      OPN   #DB_VI;  // Abro el DB a resetear
      LAR1  P##PunteroDBVI;  // Preparar el Puntero Any
      L     B#16#10;  // ID de Sintasis
      T     LB [AR1, P#0.0];
      L     B#16#2;  // Tipo de Datos
      T     LB [AR1, P#1.0];
      L     DBLG;  // Longitud del DB
      T     LW [AR1, P#2.0];
      L     DBNO;  // Numero de DB
      T     LW [AR1, P#4.0];
      L     0;
      SLW   3;
      T     LD [AR1, P#6.0];
      L     B#16#84;  // Indico el tipo DB
      T     LB [AR1, P#6.0];

      L     0;  // Que rellenar en el DB
      T     #ByteTMP;
      CALL  FILL
      ( BVAL    := #ByteTMP,
        RET_VAL := #ReturnValor,
        BLK     := #PunteroDBVI
      );  // Reseteo el DB


/////////////////////////////////////////////////////////////////////////////
// --- Reseteo - Estado del Vehiculo Inteligente

      L     0;  // Reseteo del Estado del VI
      T     #ByteTMP;
      CALL  FILL
      ( BVAL    := #ByteTMP,
        RET_VAL := #ReturnValor,
        BLK     := "DB900_Estado_Mesas".EstadoVI[#Mesa]
      );

/////////////////////////////////////////////////////////////////////////////
// --- No hay más que resetar
      JU    SistemaReset_Gestion;


/////////////////////////////////////////////////////////////////////////////
/////////////////////////////////////////////////////////////////////////////
/////////////////////////////////////////////////////////////////////////////
/////////////////////////////////////////////////////////////////////////////
// --- Reset Imposible

ResetImposible:NOP   0;
      SET;
      S     "DB840_Emision".DispoMesa[#Mesa].Protocolo.ResetNOK;  // Activacion de Reset Imposible
      R     "DB840_Emision".DispoMesa[#Mesa].Protocolo.ResetOK;  // DesActivacion de Reset OK
      R     "DB840_Emision".DispoMesa[#Mesa].Protocolo.Reset_Realizandose;  // Desactivar el Reset
      R     "DB831_Mesas".Mesas[#Mesa].Memorias.M_ResetParcial;  // Memo Reset Parcial
      R     "DB831_Mesas".Mesas[#Mesa].Memorias.M_ResetTotal;  // Memo Reset Total

      JU    SistemaReset_Gestion;


/////////////////////////////////////////////////////////////////////////////
/////////////////////////////////////////////////////////////////////////////
/////////////////////////////////////////////////////////////////////////////
/////////////////////////////////////////////////////////////////////////////
// --- Gestion de Reset
SistemaReset_Gestion:NOP   0;
      SET;
      AN    "DB840_Emision".DispoMesa[#Mesa].Protocolo.Reset_Realizandose;
      JC    SistemaReset_Fin;  // Hay Reset en el Sistema ?

      SET;
      AN    #EstadoZona.Resetear_CBx;  // Por la Zona
      AN    #EstadoZona.PerReset_CBx;
      AN    "DB841_Recepcion".DispoMesa[#Mesa].Protocolo.Reset;  // Por la Orden de la Mesa
      AN    "DB843_RecepcionPantalla".Mesa[#Mesa].Reset;  // Por la Orden de la Pantalla
      A     "DB841_Recepcion".DispoMesa[#Mesa].Protocolo.EmiOK;  // Avisado el JdT ?
      JCN   SistemaReset_Continuar;


/////////////////////////////////////////////////////////////////////////////
// --- Reset Finalizazado
      SET;
      R     "DB840_Emision".DispoMesa[#Mesa].Protocolo.Reset_Realizandose;
      R     "DB831_Mesas".Mesas[#Mesa].Memorias.M_ResetParcial;  // Memo Reset Parcial
      R     "DB831_Mesas".Mesas[#Mesa].Memorias.M_ResetTotal;  // Memo Reset Total -


/////////////////////////////////////////////////////////////////////////////
/////////////////////////////////////////////////////////////////////////////
/////////////////////////////////////////////////////////////////////////////
// --- Continuar con el Reset

SistemaReset_Continuar:NOP   0;
      SET;
      A     #FinResetTMP;  // Fin de Reset del VI ?
      S     "DB840_Emision".DispoMesa[#Mesa].Protocolo.ResetOK;  // Aviso de Fin de Reset


// --- Si no llega el Fin de Reset en un tiempo determinado
      SET;
      AN    #FinResetTMP;  // No, Fin de Reset del VI ?
      AN    "DB840_Emision".DispoMesa[#Mesa].Protocolo.ResetOK;  // No, Aviso de Fin de Reset
      AN    "DB840_Emision".DispoMesa[#Mesa].Protocolo.ResetNOK;  // No, Aviso de Fin de Reset
      A     #TIM_FinReset_OK;  // Se cumplido el tiempo de Espera
      A     "DB840_Emision".DispoMesa[#Mesa].Protocolo.Reset_Realizandose;  // Reset Realizandose
      JC    ResetImposible;  // Activar reset imposible


// --- Finalizado
      JU    SistemaReset_Fin;  // Ir al Final de Reset


/////////////////////////////////////////////////////////////////////////////
/////////////////////////////////////////////////////////////////////////////
/////////////////////////////////////////////////////////////////////////////
/////////////////////////////////////////////////////////////////////////////
// --- Fin del sistema de Reset

SistemaReset_Fin:NOP   0;
      SET;
      AN    "DB840_Emision".DispoMesa[#Mesa].Protocolo.Reset_Realizandose;
      R     "DB840_Emision".DispoMesa[#Mesa].Protocolo.ResetOK;  // No Aviso de Fin de Reset

      SET;
      A     "DB840_Emision".DispoMesa[#Mesa].Protocolo.ResetNOK;
      A     "DB841_Recepcion".DispoMesa[#Mesa].Protocolo.EmiOK;
      R     "DB840_Emision".DispoMesa[#Mesa].Protocolo.ResetNOK;  // Desactivacion de Reset Imposible



NETWORK
TITLE = ---- Presencias de la Mesa en el Reset
/////////////////////////////////////////////////////////////////////////////
// --- Presencias de la Mesa en el Reset
      SET;
      A     "DB840_Emision".Mesa[#Mesa].Protocolo.PresNormal;
      A     "DB900_Estado_Mesas".EstadoVI[#Mesa].Etapas_Reset;
      =     "DB840_Emision".Mesa[#Mesa].Protocolo.PresReset;  // Presencia de Reset

/////////////////////////////////////////////////////////////////////////////
// --- Comprobar que se esta haciendo Reset
      SET;
      AN    "DB840_Emision".DispoMesa[#Mesa].Protocolo.Reset_Realizandose;
      JC    Final_PresenciaEnReset;

/////////////////////////////////////////////////////////////////////////////
// --- Flanco en el Reset
      SET;
      A     "DB840_Emision".Mesa[#Mesa].Protocolo.PresReset;  // Emision del VI
      FP    "DB831_Mesas".Mesas[#Mesa].Memorias.MFL_PresReset;
      =     #FlancoPresReset;

/////////////////////////////////////////////////////////////////////////////
// --- Creacion de UT en Reset Total
      SET;
      A     "DB831_Mesas".Mesas[#Mesa].Memorias.M_ResetTotal;  // Memo Reset Total
      A     #FlancoPresReset;
      JCN   Final_PresenciaEnReset;

// Creo una nueva UT
      CALL  "FC723_InsertarUT_EnMesa"
      ( MesaActual := #Mesa,
        NumeroUT   := #NumeroUT
      );

      JU    Final_PresenciaEnReset;

/////////////////////////////////////////////////////////////////////////////
Final_PresenciaEnReset:NOP   0;



NETWORK
TITLE = Gestion del Control de Paro Blando
/////////////////////////////////////////////////////////////////////////////
// --- Flanco de la Activacion de la Gestion del Paro Blando
      SET;
      A     "DB841_Recepcion".DispoMesa[#Mesa].Protocolo.ParoBlando;  // Por la Orden de Mesa
      O     "DB843_RecepcionPantalla".Mesa[#Mesa].ParoBlando;  // Por la Orden de la Pantalla
      FP    "DB831_Mesas".Mesas[#Mesa].Memorias.MFL_ParoBlando;  // Memo Paro Blando - Pos: 22.7
      =     #FlancoParoBlando;

      SET;
      A     #FinParoBlando;  // No hace caso si no hay Paro Blando
      A     "DB900_Estado_Mesas".EstadoVI[#Mesa].Paro_Blando;
      A     "DB840_Emision".DispoMesa[#Mesa].Protocolo.ParoBlando_Realizandose;
      =     #FinParoBlandoTMP;


/////////////////////////////////////////////////////////////////////////////
// --- Activacion de la Gestion del Paro Blando

      AN    #FlancoParoBlando;
      JC    SistemaParoBlando_Gestion;  // Hay que realizar el Paro Blando ?

      SET;
      S     "DB840_Emision".DispoMesa[#Mesa].Protocolo.ParoBlando_Realizandose;

      JU    SistemaParoBlando_Gestion;

/////////////////////////////////////////////////////////////////////////////
/////////////////////////////////////////////////////////////////////////////
/////////////////////////////////////////////////////////////////////////////
/////////////////////////////////////////////////////////////////////////////
// --- Paro Blando Imposible

ParoBlandoImposible:NOP   0;
      S     "DB840_Emision".DispoMesa[#Mesa].Protocolo.ParoBlandoNOK;  // Activacion de Paro Blando Imposible
      R     "DB840_Emision".DispoMesa[#Mesa].Protocolo.ParoBlandoOK;  // DesActivacion de Paro Blando OK

      R     "DB840_Emision".DispoMesa[#Mesa].Protocolo.ParoBlando_Realizandose;  // Acabado Paro Blando
      R     "DB840_Emision".DispoMesa[#Mesa].Protocolo.Marcha;  // Se pasa a Paro
      S     "DB840_Emision".DispoMesa[#Mesa].Protocolo.Paro;

      JU    SistemaParoBlando_Gestion;

/////////////////////////////////////////////////////////////////////////////
/////////////////////////////////////////////////////////////////////////////
/////////////////////////////////////////////////////////////////////////////
// --- Gestion del Paro Blando

SistemaParoBlando_Gestion:NOP   0;
      SET;
      AN    "DB840_Emision".DispoMesa[#Mesa].Protocolo.ParoBlando_Realizandose;
      JC    SistemaParoBlando_Fin;  // Hay Paro Blando en el Sistema ?

      SET;
      AN    "DB841_Recepcion".DispoMesa[#Mesa].Protocolo.ParoBlando;  // Por la Orden de la Mesa
      AN    "DB843_RecepcionPantalla".Mesa[#Mesa].ParoBlando;  // Por la Orden de la Pantalla
      A     "DB841_Recepcion".DispoMesa[#Mesa].Protocolo.EmiOK;  // Avisado el JdT ?
      JCN   SistemaParoBlando_Continuar;


/////////////////////////////////////////////////////////////////////////////
/////////////////////////////////////////////////////////////////////////////
/////////////////////////////////////////////////////////////////////////////
// --- Fin de Paro Blando Finalizado

      SET;
      R     "DB840_Emision".DispoMesa[#Mesa].Protocolo.ParoBlando_Realizandose;  // Acabado Paro Blando
      R     "DB840_Emision".DispoMesa[#Mesa].Protocolo.Marcha;  // Se pasa a Paro
      S     "DB840_Emision".DispoMesa[#Mesa].Protocolo.Paro;

/////////////////////////////////////////////////////////////////////////////
/////////////////////////////////////////////////////////////////////////////
/////////////////////////////////////////////////////////////////////////////
// --- Continuar con el Paro Blando
SistemaParoBlando_Continuar:NOP   0;

      SET;
      A     #FinParoBlandoTMP;  // Fin de ParoBlando del VI ?
      S     "DB840_Emision".DispoMesa[#Mesa].Protocolo.ParoBlandoOK;  // Aviso de Fin de Paro Blando

// --- Si no llega el Fin de Paro Blando en un tiempo determinado
      SET;
      AN    #FinParoBlandoTMP;  // No, Fin de Paro Blando del VI ?
      AN    "DB840_Emision".DispoMesa[#Mesa].Protocolo.ParoBlandoOK;  // No, Aviso de Fin de Paro Blando
      AN    "DB840_Emision".DispoMesa[#Mesa].Protocolo.ParoBlandoNOK;  // No, Aviso de Fin de Paro Blando
      A     #TIM_FinParoBlando_OK;  // Se cumplido el tiempo de Espera
      A     "DB840_Emision".DispoMesa[#Mesa].Protocolo.ParoBlando_Realizandose;  // Paro Blando Realizandose
      JC    ParoBlandoImposible;  // Activar Paro Blando imposible


/////////////////////////////////////////////////////////////////////////////
// --- Fin del sistema de Paro Blando

SistemaParoBlando_Fin:NOP   0;
      SET;
      AN    "DB840_Emision".DispoMesa[#Mesa].Protocolo.ParoBlando_Realizandose;
      R     "DB840_Emision".DispoMesa[#Mesa].Protocolo.ParoBlandoOK;  // No Aviso de Fin de Paro Blando

      SET;
      A     "DB840_Emision".DispoMesa[#Mesa].Protocolo.ParoBlandoNOK;
      A     "DB841_Recepcion".DispoMesa[#Mesa].Protocolo.EmiOK;
      R     "DB840_Emision".DispoMesa[#Mesa].Protocolo.ParoBlandoNOK;  // Desactivacion de Paro Blando Imposible



NETWORK
TITLE = Gestion del Control de Error de la Mesa
/////////////////////////////////////////////////////////////////////////////
// --- Calculo del Error de la Mesa

      AN    "DB900_Estado_Mesas".EstadoVI[#Mesa].Error_Mx;
      JC    NoErrorEnMesa;


/////////////////////////////////////////////////////////////////////////////
      L     #Mesa;  // Puntero al DB de Estado VI
      L     "CTE_Long_VIMesa";  // Longitud de la UDT 20
      *D;
      SLD   3;
      T     #P_EstadoVI;

      L     "CTE_NDB_EstadoVIMesa";  // DB de Estado VI
      T     #DBEstadoVI;

      L     #P_EstadoVI;  // Punteros
      L     P#2.0;
      +D;
      LAR2;
      T     #PunteroDBTMP;  // Offset dentro del DB

      OPN   DB [#DBEstadoVI];
Bucle_ErrorVI:NOP   0;
      A     DBX [AR2, P#0.0];
      JC    EncontradoErrorEnMesa;

      +AR2  P#0.1;
      JU    Bucle_ErrorVI;


/////////////////////////////////////////////////////////////////////////////
// --- Con Error
EncontradoErrorEnMesa:NOP   0;
      TAR2;
      L     #PunteroDBTMP;
      -D;
      L     1;
      +D;
      T     #NumeroErrorVI;
      T     "DB840_Emision".DispoMesa[#Mesa].Error;

      L     #NumeroErrorVI;
      T     #CodigoErrorMesa;
      T     "DB861_FIFO_Errores".Mesas[#Mesa];

      JU    FinGestion_Error;


/////////////////////////////////////////////////////////////////////////////
// --- Sin Error
NoErrorEnMesa:NOP   0;
      L     0;
      T     #CodigoErrorMesa;
      T     "DB840_Emision".DispoMesa[#Mesa].Error;
      T     "DB861_FIFO_Errores".Mesas[#Mesa];

      JU    FinGestion_Error;


/////////////////////////////////////////////////////////////////////////////
// --- Rearme y Activacion del Error
FinGestion_Error:NOP   0;
      SET;
      A     #EstadoZona.Rearme_CBx;  // Por la Zona
      O     #RearmeError;  // Manualmente (Exterior)
      O     "DB841_Recepcion".DispoMesa[#Mesa].Protocolo.Rearme;  // Por la Orden
      O     "DB843_RecepcionPantalla".Mesa[#Mesa].Rearme;  // Por la Orden de Pantalla
      =     "DB902_Estado_ZonaMesa".EstadoMesas[#Mesa].Rearme_CBx;

      SET;
      A     "DB900_Estado_Mesas".EstadoVI[#Mesa].Error_Mx;
      =     "DB840_Emision".DispoMesa[#Mesa].Protocolo.Error;  // Esta en Error el VI



REGION Network 10: Cierre del Protocolo de la Mesa
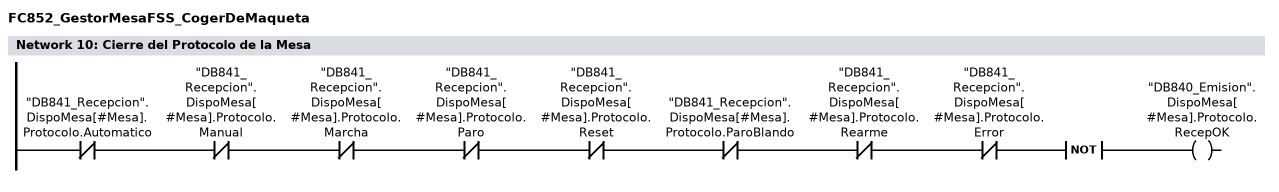
   RUNG wire#powerrail
      I_Contact( "DB841_Recepcion".DispoMesa[#Mesa].Protocolo.Automatico )
      I_Contact( "DB841_Recepcion".DispoMesa[#Mesa].Protocolo.Manual )
      I_Contact( "DB841_Recepcion".DispoMesa[#Mesa].Protocolo.Marcha )
      I_Contact( "DB841_Recepcion".DispoMesa[#Mesa].Protocolo.Paro )
      I_Contact( "DB841_Recepcion".DispoMesa[#Mesa].Protocolo.Reset )
      I_Contact( "DB841_Recepcion".DispoMesa[#Mesa].Protocolo.ParoBlando )
      I_Contact( "DB841_Recepcion".DispoMesa[#Mesa].Protocolo.Rearme )
      I_Contact( "DB841_Recepcion".DispoMesa[#Mesa].Protocolo.Error )
      Not()
      Coil( "DB840_Emision".DispoMesa[#Mesa].Protocolo.RecepOK )
   END_RUNG
   // the same network as SCL:
   "DB840_Emision".DispoMesa[#Mesa].Protocolo.RecepOK := NOT (NOT "DB841_Recepcion".DispoMesa[#Mesa].Protocolo.Automatico AND NOT "DB841_Recepcion".DispoMesa[#Mesa].Protocolo.Manual AND NOT "DB841_Recepcion".DispoMesa[#Mesa].Protocolo.Marcha AND NOT "DB841_Recepcion".DispoMesa[#Mesa].Protocolo.Paro AND NOT "DB841_Recepcion".DispoMesa[#Mesa].Protocolo.Reset AND NOT "DB841_Recepcion".DispoMesa[#Mesa].Protocolo.ParoBlando AND NOT "DB841_Recepcion".DispoMesa[#Mesa].Protocolo.Rearme AND NOT "DB841_Recepcion".DispoMesa[#Mesa].Protocolo.Error);
END_REGION

NETWORK
TITLE = Cierre del Protocolo de la Pantalla
/////////////////////////////////////////////////////////////////////////////
// --- Cierre del protocolo de las ordenes de la Pantalla
// --- Doy por tratada la Orden

      L     0;  // Que rellenar en el DB
      T     #ByteTMP;

      CALL  FILL
      ( BVAL    := #ByteTMP,
        RET_VAL := #ReturnValor,
        BLK     := "DB843_RecepcionPantalla".Mesa[#Mesa]
      );  // Reseteo el la zona temp



NETWORK
TITLE = Actualizacion del Estado para el Vehiculo Inteligente
/////////////////////////////////////////////////////////////////////////////
// --- Trasvase - Estado de la Mesa para VI

      A     "DB840_Emision".DispoMesa[#Mesa].Protocolo.Error;
      =     "DB902_Estado_ZonaMesa".EstadoMesas[#Mesa].Error_CBx;
      A     "DB840_Emision".DispoMesa[#Mesa].Protocolo.Marcha;
      =     "DB902_Estado_ZonaMesa".EstadoMesas[#Mesa].Marcha_CBx;
      A     "DB840_Emision".DispoMesa[#Mesa].Protocolo.Paro;
      =     "DB902_Estado_ZonaMesa".EstadoMesas[#Mesa].Paro_CBx;

      A     "DB840_Emision".DispoMesa[#Mesa].Protocolo.Automatico;
      =     "DB902_Estado_ZonaMesa".EstadoMesas[#Mesa].Automatico_CBx;
      A     "DB840_Emision".DispoMesa[#Mesa].Protocolo.Manual;
      =     "DB902_Estado_ZonaMesa".EstadoMesas[#Mesa].Manual_CBx;

      A     #FlancoReset;
      =     "DB902_Estado_ZonaMesa".EstadoMesas[#Mesa].Resetear_CBx;
      A     "DB840_Emision".DispoMesa[#Mesa].Protocolo.Reset_Realizandose;
      =     "DB902_Estado_ZonaMesa".EstadoMesas[#Mesa].PerReset_CBx;

      A     "DB840_Emision".DispoMesa[#Mesa].Protocolo.ParoBlando_Realizandose;
      =     "DB902_Estado_ZonaMesa".EstadoMesas[#Mesa].ParoBlando_CBx;



NETWORK
TITLE = Control de Error de Mesa por Orden del JdT
/////////////////////////////////////////////////////////////////////////////
/////////////////////////////////////////////////////////////////////////////
// --- Rearme de Errores Generados
// --- Borrado errores Mesa --> JdT

      SET;
      A     #EstadoZona.Rearme_CBx;  // Por la Zona
      O     #RearmeError;  // Manualmente (Exterior)
      O     "DB841_Recepcion".DispoMesa[#Mesa].Protocolo.Rearme;  // Por la Orden
      O     "DB843_RecepcionPantalla".Mesa[#Mesa].Rearme;  // Por la Orden de Pantalla
      JCN   NoRearme_ErrorJdT;

      SET;
      R     "DB900_Estado_Mesas".EstadoVI[#Mesa].Err_EnviadoPorJDT;  // Error Enviado por JDT
      R     "DB900_Estado_Mesas".EstadoVI[#Mesa].Error_Mx;  // Error de Mesa


NoRearme_ErrorJdT:NOP   0;


/////////////////////////////////////////////////////////////////////////////
/////////////////////////////////////////////////////////////////////////////
// --- Mirar errores Mesa --> JdT

      SET;
      AN    "DB841_Recepcion".DispoMesa[#Mesa].Protocolo.Error;
      JC    NoRecibido_ErrorJdT;

      SET;
      S     "DB900_Estado_Mesas".EstadoVI[#Mesa].Err_EnviadoPorJDT;  // Error Enviado por JDT
      S     "DB900_Estado_Mesas".EstadoVI[#Mesa].Error_Mx;  // Error de Mesa

NoRecibido_ErrorJdT:NOP   0;



NETWORK
TITLE = Control de Errores entre la Mesa y el Tracking
/////////////////////////////////////////////////////////////////////////////
/////////////////////////////////////////////////////////////////////////////
/////////////////////////////////////////////////////////////////////////////
// --- Rearme de Errores Generados
// --- Borrado errores Mesa --> Tracking

      SET;
      A     #EstadoZona.Rearme_CBx;  // Por la Zona
      O     #RearmeError;  // Manualmente (Exterior)
      O     "DB841_Recepcion".DispoMesa[#Mesa].Protocolo.Rearme;  // Por la Orden
      O     "DB843_RecepcionPantalla".Mesa[#Mesa].Rearme;  // Por la Orden de Pantalla
      JCN   NoRearme_ErrorTracking;

      SET;
      R     "DB900_Estado_Mesas".EstadoVI[#Mesa].Err_DatosPLC;  // Error Datos del PLC
      R     "DB900_Estado_Mesas".EstadoVI[#Mesa].Error_Mx;  // Error de Mesa


NoRearme_ErrorTracking:NOP   0;


/////////////////////////////////////////////////////////////////////////////
/////////////////////////////////////////////////////////////////////////////
/////////////////////////////////////////////////////////////////////////////
// --- Listado de Errores implementados:
// ---     * Mesa Vacia con existencia de una UT
// ---     * Mesa Ocupada sin existencia de una UT

      CALL  "FC870_MesaSinUT"
      ( Mesa  := #Mesa,
        SinUT := #SinUT_EnMesa
      );

      SET;
      AN    "DB850_DefinicionMesas".Mesa[#Mesa].ConfigMesa.SinErrorDeDatosVacia;
      A     "DB840_Emision".DispoMesa[#Mesa].Protocolo.Marcha;
      AN    "DB840_Emision".DispoMesa[#Mesa].Protocolo.Error;
      A     "DB900_Estado_Mesas".EstadoVI[#Mesa].Etapa_Vacia;
      AN    #SinUT_EnMesa;
      =     #ErrorMesaVacia;

      SET;
      AN    "DB850_DefinicionMesas".Mesa[#Mesa].ConfigMesa.SinErrorDeDatosCargada;
      A     "DB840_Emision".DispoMesa[#Mesa].Protocolo.Marcha;
      AN    "DB840_Emision".DispoMesa[#Mesa].Protocolo.Error;
      A     "DB900_Estado_Mesas".EstadoVI[#Mesa].Etapa_Cargada;
      A     #SinUT_EnMesa;
      =     #ErrorMesaOcupada;

      SET;
      A     #ErrorMesaVacia;
      O     #ErrorMesaOcupada;
      =     #ActivarTMPErrorMesa;


/////////////////////////////////////////////////////////////////////////////
// ---     * Esperar tiempo antes de activar el Error

      CALL  "FC899_TMP"
      ( Temporizar     := #ActivarTMPErrorMesa,
        Valor_Tiempo   := 20,
        Base_tiempo_ms := 1000,
        Tiempo_OK      := #TIM_ErrorMesa_OK,
        Valor_Actual   := "DB831_Mesas".Mesas[#Mesa].TMP_ErrorDatos
      );


/////////////////////////////////////////////////////////////////////////////
// --- Mirar errores Mesa --> Tracking
      SET;
      AN    #TIM_ErrorMesa_OK;
      JC    NoExiste_ErrorTracking;

      SET;
      S     "DB900_Estado_Mesas".EstadoVI[#Mesa].Err_DatosPLC;  // Error Datos del PLC
      S     "DB900_Estado_Mesas".EstadoVI[#Mesa].Error_Mx;  // Error de Mesa

NoExiste_ErrorTracking:NOP   0;



NETWORK
TITLE = Cambio de Mesa o creación de la UT -- DIstribucion
// Realiza:
//  - Gestion de la realización del cambio de Mesa de la UT
//  - Creación de la UT nueva
/////////////////////////////////////////////////////////////////////////////
// --- Distribución de lo que se HARA ? y CUANDO ?
/////////////////////////////////////////////////////////////////////////////
// --- Entrada de la UT por E0
// --- Entrada de la UT por E1
// --- Entrada de la UT por E2
// --- Entrada de la UT por E3
// --- Entrada de la UT por E4
// ---
// --- Nota: Hay que identificar en cada entrada dos casos:
// ---       Cuando cambia de Mesa - Codigo 11
// ---       Cuando se crea la UT  - Codigo 12
/////////////////////////////////////////////////////////////////////////////

      SET;
      A     #TransferirUT;  // Orden de Transferir la UT
      FP    "DB831_Mesas".Mesas[#Mesa].Memorias.MFL_TransferirUT;
      =     #FlancoTransferirUT;

      SET;
      AN    #FlancoTransferirUT;
      JC    FinalControlUTs_EnMesa;


/////////////////////////////////////////////////////////////////////////////
/////////////////////////////////////////////////////////////////////////////
// ---                     DISTRIBUCION
/////////////////////////////////////////////////////////////////////////////
/////////////////////////////////////////////////////////////////////////////

      SET;  //  Entrada E00
      A     "DB900_Estado_Mesas".EstadoVI[#Mesa].Etapas_Carga_E0;
      A     #FlancoTransferirUT;
      JC    Caso_EntradaE0;

      SET;  //  Entrada E01
      A     "DB900_Estado_Mesas".EstadoVI[#Mesa].Etapas_Carga_E1;
      A     #FlancoTransferirUT;
      JC    Caso_EntradaE1;

      SET;  //  Entrada E02
      A     "DB900_Estado_Mesas".EstadoVI[#Mesa].Etapas_Carga_E2;
      A     #FlancoTransferirUT;
      JC    Caso_EntradaE2;

      SET;  //  Entrada E03
      A     "DB900_Estado_Mesas".EstadoVI[#Mesa].Etapas_Carga_E3;
      A     #FlancoTransferirUT;
      JC    Caso_EntradaE3;

      SET;  //  Entrada E04
      A     "DB900_Estado_Mesas".EstadoVI[#Mesa].Etapas_Carga_E4;
      A     #FlancoTransferirUT;
      JC    Caso_EntradaE4;

/////////////////////////////////////////////////////////////////////////////
// ---- No hay que hacer nada todavia

      JU    FinalControlUTs_EnMesa;



/////////////////////////////////////////////////////////////////////////////
/////////////////////////////////////////////////////////////////////////////
// ---                   FIN DE LA DISTRIBUCION
/////////////////////////////////////////////////////////////////////////////
/////////////////////////////////////////////////////////////////////////////


/////////////////////////////////////////////////////////////////////////////
/////////////////////////////////////////////////////////////////////////////
// ---    Caso 0: En la Entrada E00
// ---    * Siempre hay que crear UT en la mesa

Caso_EntradaE0:NOP   0;
      JU    CrearUT_EnMesa;  // Siempre crear UT en la Mesa


/////////////////////////////////////////////////////////////////////////////
/////////////////////////////////////////////////////////////////////////////
// ---    Caso: En la Entrada E01
// ---    * Si No Definada Mesa - Crear UT
// ---    * Si Definida Mesa - Recoger UT de la Mesa Definida

Caso_EntradaE1:NOP   0;
      L     #Mesa_E01;  // Mesa E01 = 0
      L     0;  // No se puede traer de otra Mesa la UT
      ==I;
      JC    CrearUT_EnMesa;

// ------------ Cuando hay que Cambiar de Mesa la UT

      L     #Mesa_E01;
      T     #MesaDeCambio;

      JU    CambioDeUTs_EnMesa;  // Se acabo


/////////////////////////////////////////////////////////////////////////////
/////////////////////////////////////////////////////////////////////////////
// ---    Caso: En la Entrada E02
// ---    * Si No Definada Mesa - Crear UT
// ---    * Si Definida Mesa - Recoger UT de la Mesa Definida

Caso_EntradaE2:NOP   0;
      L     #Mesa_E02;  // Mesa E01 = 0
      L     0;  // No se puede traer de otra Mesa la UT
      ==I;
      JC    CrearUT_EnMesa;

// ------------ Cuando hay que Cambiar de Mesa la UT

      L     #Mesa_E02;
      T     #MesaDeCambio;

      JU    CambioDeUTs_EnMesa;  // Se acabo


/////////////////////////////////////////////////////////////////////////////
/////////////////////////////////////////////////////////////////////////////
// ---    Caso: En la Entrada E03
// ---    * Si No Definada Mesa - Crear UT
// ---    * Si Definida Mesa - Recoger UT de la Mesa Definida

Caso_EntradaE3:NOP   0;
      L     #Mesa_E03;  // Mesa E01 = 0
      L     0;  // No se puede traer de otra Mesa la UT
      ==I;
      JC    CrearUT_EnMesa;

// ------------ Cuando hay que Cambiar de Mesa la UT

      L     #Mesa_E03;
      T     #MesaDeCambio;

      JU    CambioDeUTs_EnMesa;  // Se acabo


/////////////////////////////////////////////////////////////////////////////
/////////////////////////////////////////////////////////////////////////////
// ---    Caso: En la Entrada E04
// ---    * Si No Definada Mesa - Crear UT
// ---    * Si Definida Mesa - Recoger UT de la Mesa Definida

Caso_EntradaE4:NOP   0;
      L     #Mesa_E04;  // Mesa E01 = 0
      L     0;  // No se puede traer de otra Mesa la UT
      ==I;
      JC    CrearUT_EnMesa;

// ------------ Cuando hay que Cambiar de Mesa la UT

      L     #Mesa_E04;
      T     #MesaDeCambio;

      JU    CambioDeUTs_EnMesa;  // Se acabo



NETWORK
TITLE = -- Cambio de Mesa
/////////////////////////////////////////////////////////////////////////////
/////////////////////////////////////////////////////////////////////////////
/////////////////////////////////////////////////////////////////////////////
// ---    Cambiar de Mesa la UT
CambioDeUTs_EnMesa:NOP   0;

      L     10;  // Tipo de Carga = Bandeja Pequeña
      T     #BandejaPequeña;

/////////////////////////////////////////////////////////////////////////////
// --- FASE01 :  Primera UT --> Hay Que Cambiar de Mesa ?
ControlCambiarUT01:NOP   0;
      L     "DB810_ColasMesas".Colas[#MesaDeCambio].UT_PrimeraMesa;
      T     #NumeroUT;

      L     #NumeroUT;
      L     0;  // No existe UT
      ==I;
      JC    FinalControlUTs_EnMesa;

// --- 1.1. >>> Si MesaActual <> 0 --> Cambiar de Mesa la 1º UT
      L     "DB812_UTs_Control".UT[#NumeroUT].MesaDestino;
      L     0;
      ==I;
      JC    ControlCambiarUT02;


// --- 1.2. >>> Si MesaActual <> Destino --> Cambiar de Mesa la 1º UT
      L     "DB812_UTs_Control".UT[#NumeroUT].MesaActual;
      L     "DB812_UTs_Control".UT[#NumeroUT].MesaDestino;
      ==I;
      JC    ControlCambiarUT02;


// --- 1.3. >>> Hay que Cambiar de Mesa
      CALL  "FC724_CambiarUT_DeMesa"
      ( NumeroUT    := #NumeroUT,
        NuevaMesa   := #Mesa,
        AlPrincipio := "DB850_DefinicionMesas".Mesa[#Mesa].ConfigMesa.MeterAlPrincipio
      );  // Cambia la UT a la Nueva Mesa

      L     0;  // Es de Ordenes Especiales - Resetear
      T     "DB812_UTs_Control".UT[#NumeroUT].EstadoRecepcionUT;
      T     "DB812_UTs_Control".UT[#NumeroUT].EstadoEventoRecibido;
      L     11;  // Aviso de Cambio de Mesa de la UT
      T     "DB812_UTs_Control".UT[#NumeroUT].EstadoEmisionUT;


// --- 1.4. >>> Es Doble Pequeña
      SET;  // En Mesa Activo la Doble Pequeña
      AN    #ActivarDoblePequeña;
      JC    FinalControlUTs_EnMesa;

      SET;  // Es Doble Pequeña ?
      AN    "DB812_UTs_Control".UT[#NumeroUT].AtributosDeLaUT.LadoDeLaEtiqueta;
      JC    FinalControlUTs_EnMesa;


// --- 1.5. >>> Hay que Cambiar Dos UTs, Hay doble Pequeña
      L     "DB810_ColasMesas".Colas[#MesaDeCambio].UT_PrimeraMesa;
      T     #NumeroUT;

      L     #NumeroUT;
      L     0;  // No existe UT
      ==I;
      JC    FinalControlUTs_EnMesa;

      CALL  "FC724_CambiarUT_DeMesa"
      ( NumeroUT    := #NumeroUT,
        NuevaMesa   := #Mesa,
        AlPrincipio := "DB850_DefinicionMesas".Mesa[#Mesa].ConfigMesa.MeterAlPrincipio
      );  // Cambia la UT a la Nueva Mesa

      L     0;  // Es de Ordenes Especiales - Resetear
      T     "DB812_UTs_Control".UT[#NumeroUT].EstadoRecepcionUT;
      T     "DB812_UTs_Control".UT[#NumeroUT].EstadoEventoRecibido;
      L     11;  // Aviso de Cambio de Mesa de la UT
      T     "DB812_UTs_Control".UT[#NumeroUT].EstadoEmisionUT;

      JU    FinalControlUTs_EnMesa;


/////////////////////////////////////////////////////////////////////////////
// --- FASE02 : Segunda UT --> Hay Que Cambiar de Mesa ?
ControlCambiarUT02:NOP   0;
      L     "DB812_UTs_Control".UT[#NumeroUT].UT_SiguienteMesa;
      T     #NumeroUT;

      L     #NumeroUT;
      L     0;  // No existe UT
      ==I;
      JC    FinalControlUTs_EnMesa;

// --- 2.2. >>> Si MesaActual <> 0 --> Cambiar de Mesa la 2º UT
      L     "DB812_UTs_Control".UT[#NumeroUT].MesaDestino;
      L     0;
      ==I;
      JC    FinalControlUTs_EnMesa;


// --- 2.2. >>> Si MesaActual <> Destino --> Cambiar de Mesa la 2º UT
      L     "DB812_UTs_Control".UT[#NumeroUT].MesaActual;
      L     "DB812_UTs_Control".UT[#NumeroUT].MesaDestino;
      ==I;
      JC    FinalControlUTs_EnMesa;


// --- 2.3. >>> Hay que Cambiar de Mesa
      CALL  "FC724_CambiarUT_DeMesa"
      ( NumeroUT    := #NumeroUT,
        NuevaMesa   := #Mesa,
        AlPrincipio := "DB850_DefinicionMesas".Mesa[#Mesa].ConfigMesa.MeterAlPrincipio
      );  // Cambia la UT a la Nueva Mesa

      L     0;  // Es de Ordenes Especiales - Resetear
      T     "DB812_UTs_Control".UT[#NumeroUT].EstadoRecepcionUT;
      T     "DB812_UTs_Control".UT[#NumeroUT].EstadoEventoRecibido;
      L     11;  // Aviso de Cambio de Mesa de la UT
      T     "DB812_UTs_Control".UT[#NumeroUT].EstadoEmisionUT;

      JU    FinalControlUTs_EnMesa;



NETWORK
TITLE = -- Creación de la UT
/////////////////////////////////////////////////////////////////////////////
/////////////////////////////////////////////////////////////////////////////
/////////////////////////////////////////////////////////////////////////////
// ---    Creacion de la UT
// ---    * Insertar una nueva UT en la Mesa
// ---    * Aviso de Nueva UT en la Mesa - Codigo 12
CrearUT_EnMesa:NOP   0;

      CALL  "FC723_InsertarUT_EnMesa"
      ( MesaActual := #Mesa,
        NumeroUT   := #NumeroUT
      );

      L     12;  // Aviso de Nueva UT en la Mesa
      T     "DB812_UTs_Control".UT[#NumeroUT].EstadoEmisionUT;

      JU    FinalControlUTs_EnMesa;

// --- Fin de la Creacion de la UT
/////////////////////////////////////////////////////////////////////////////
/////////////////////////////////////////////////////////////////////////////
/////////////////////////////////////////////////////////////////////////////



NETWORK
TITLE = -- Final (Cambio de Mesa o creación de la UT)
/////////////////////////////////////////////////////////////////////////////
/////////////////////////////////////////////////////////////////////////////
/////////////////////////////////////////////////////////////////////////////
// --- Fin del Segmento

FinalControlUTs_EnMesa:NOP   0;



NETWORK
TITLE = Introducir los Datos para el Scada
/////////////////////////////////////////////////////////////////////////////
      CALL  "FC960_ScadaMesa"
      ( NumMesa := #Mesa
      );


END_FUNCTION

FUNCTION "FC860_Informe_DatosUT" : Void   // FC860, STL
{ S7_Optimized_Access := 'FALSE' }
// stored: AutoNumber false
   VAR_INPUT
      Mesa : UInt;
   END_VAR
   VAR_OUTPUT
      Informe_DatosUT : "UDT_Informe_DatosUT";
   END_VAR
   VAR_TEMP
      NumeroUT : Int;
      Relleno : Byte;
      ValorReturn : Int;
   END_VAR
BEGIN

NETWORK
TITLE = Inicializar
//////////////////////////////////////////////////////////////////////
/// Inicializar Variables

      L     0;
      T     #Relleno;

      CALL  FILL
      ( BVAL    := #Relleno,
        RET_VAL := #ValorReturn,
        BLK     := #Informe_DatosUT
      );



NETWORK
TITLE = Buscar Primera UT de la Mesa
//////////////////////////////////////////////////////////////////////
/// Buscar Primera UT de la Mesa
      L     "DB810_ColasMesas".Colas[#Mesa].UT_PrimeraMesa;
      T     #NumeroUT;

      L     #NumeroUT;
      L     0;
      <>I;
      JC    CrearInforme;

      BE;  // - Finalizar bloque



NETWORK
TITLE = Crear Informe
CrearInforme:NOP   0;

//////////////////////////////////////////////////////////////////////
/// Crear Informe de la UT

      L     "DB812_UTs_Control".UT[#NumeroUT].MesaDestino;
      T     #Informe_DatosUT.MesaDestino;

      L     "DB812_UTs_Control".UT[#NumeroUT].TipoCarga;
      T     #Informe_DatosUT.TipoCarga;

      SET;
      A     "DB812_UTs_Control".UT[#NumeroUT].AtributosDelaCarga.Vacia;
      =     #Informe_DatosUT.AtributosCarga.Vacia;
      SET;
      A     "DB812_UTs_Control".UT[#NumeroUT].AtributosDelaCarga.Pila;
      =     #Informe_DatosUT.AtributosCarga.Pila;
      SET;
      A     "DB812_UTs_Control".UT[#NumeroUT].AtributosDelaCarga.Remontada;
      =     #Informe_DatosUT.AtributosCarga.Remontada;


      L     "DB815_UTs_Datos".UT[#NumeroUT].CodigoEnfardado;
      T     #Informe_DatosUT.Enfradado;
      L     "DB815_UTs_Datos".UT[#NumeroUT].CodigoFlejado;
      T     #Informe_DatosUT.Flejado;
      L     "DB815_UTs_Datos".UT[#NumeroUT].CodigoEtiquetado;
      T     #Informe_DatosUT.Etiquetado;

      L     "DB815_UTs_Datos".UT[#NumeroUT].CotaAltura;
      T     #Informe_DatosUT.CotaAltura;
      L     "DB815_UTs_Datos".UT[#NumeroUT].CotaAnchura;
      T     #Informe_DatosUT.CotaAnchura;
      L     "DB815_UTs_Datos".UT[#NumeroUT].CotaProfundidad;
      T     #Informe_DatosUT.CotaLargura;

      L     "DB815_UTs_Datos".UT[#NumeroUT].Peso;
      T     #Informe_DatosUT.Peso;

      SET;
      A     "DB812_UTs_Control".UT[#NumeroUT].AtributosDeLaUT.LadoDeLaEtiqueta;
      =     #Informe_DatosUT.PosEtiqueta.Derecha;

      SET;
      AN    "DB812_UTs_Control".UT[#NumeroUT].AtributosDeLaUT.LadoDeLaEtiqueta;
      =     #Informe_DatosUT.PosEtiqueta.Izquierda;

// nieves añadido volcado de la información de las etiquetas

      CALL  MOVE
      ( IN  := "DB814_UTs_Etiqueta".UT[#NumeroUT].Etiqueta,
        OUT := #Informe_DatosUT.etiqueta
      );


      L     "DB814_UTs_Etiqueta".UT[#NumeroUT].EtiquetaRouter;
      T     #Informe_DatosUT.EtiquetaRouter;

// fin añadido nieves
      BE;  // - Finalizar bloque


END_FUNCTION

FUNCTION "FC876_BorrarEstructura" : Void   // FC876, LAD
TITLE = BorrarEstructura
{ S7_Optimized_Access := 'FALSE' }
AUTHOR : TRACKING
NAME : 20130301
VERSION : 3.0
// Borra un numero de bytes de un DB desde Offset que se indique
// stored: AutoNumber false, SetENOAutomatically false
   VAR_INPUT
      NumDB : Word;   // Numero del DB
      POffset : DWord;   // Puntero del Offset dento del DB
      NumBytes : UInt;   // Numero de Bytes que hay que borrar
   END_VAR
   VAR_TEMP
      Guardar_AR1 : DWord;
      Guardar_AR2 : DWord;
      PAny_DB : Any;
      ReturnValor : Int;
      Cero : Byte;
   END_VAR
BEGIN

NETWORK
TITLE = Inicializar Punteros Any
//////////////////////////////////////////////////////////////////////////////
//////////////////////////////////////////////////////////////////////////////
/// Tareas Iniciales

      TAR1  #Guardar_AR1;  // Guardar AR1 y AR2
      TAR2  #Guardar_AR2;


//////////////////////////////////////////////////////////////////////////////
//////////////////////////////////////////////////////////////////////////////
/// Puntero Any Origen

      LAR2  P##PAny_DB;  // - Any - DB de Origen
      L     B#16#10;  //   10H para S7
      T     LB [AR2, P#0.0];
      L     B#16#2;  //   Tipo de Datos (BYTE)
      T     LB [AR2, P#1.0];
      L     #NumBytes;  //   Cantidad de datos
      T     LW [AR2, P#2.0];
      L     #NumDB;  //   Numero de DB
      T     LW [AR2, P#4.0];
      L     #POffset;  //   Direccion de Inicio
      T     LD [AR2, P#6.0];
      L     B#16#84;  //   El Area de Memoria = DB (Nota: No 84)
      T     LB [AR2, P#6.0];


//////////////////////////////////////////////////////////////////////////////
//////////////////////////////////////////////////////////////////////////////
/// Tareas Finales

      LAR1  #Guardar_AR1;  // Recuperar AR1 y AR2
      LAR2  #Guardar_AR2;



NETWORK
TITLE = Borrado
//////////////////////////////////////////////////////////////////////////////
//////////////////////////////////////////////////////////////////////////////
/// Borrrado de los Datos

      L     0;
      T     #Cero;

      CALL  FILL
      ( BVAL    := #Cero,
        RET_VAL := #ReturnValor,
        BLK     := #PAny_DB
      );  // Inicializo las Entradas



END_FUNCTION

FUNCTION "FC883_CalcularError_Armarios" : Void   // FC883, LAD
{ S7_Optimized_Access := 'FALSE' }
AUTHOR : ERRORES
NAME : 20160407
VERSION : 3.1
// stored: AutoNumber false, SetENOAutomatically false
   VAR_INPUT
      NumDB_Errores : UInt;
      Numero : UInt;
   END_VAR
   VAR_IN_OUT
      Codigo : UDInt;
      Emergencia : Bool;
      ErrorGrave : Bool;
      ErrorLeve : Bool;
   END_VAR
   VAR_TEMP
      ErrorFIFO : UDInt;
      P_Inicial : DWord;
      P_Final : DWord;
      NumDB : Word;
      Armario : UDInt;
      NumEmerg : UDInt;
      NumErrorGrave : UDInt;
      NumErrorLeve : UDInt;
      OffsetEmerg : UInt;
      OffsetErrorGrave : UInt;
      OffsetErrorLeve : UInt;
      MaxBitsGraves : UInt;
      MaxBitsLeves : UInt;
      LongBits : UInt;
      Zona : UInt;
   END_VAR
BEGIN

NETWORK
TITLE = Inicializar
///////////////////////////////////////////////////////////////////////////
// --- Inicializar Variables

      L     #NumDB_Errores;  // DB de Errores FIFO
      T     #NumDB;

      L     0;
      T     #NumEmerg;  // nieves 28/08/25      // No hay Emergencia (Inicial)
      T     #NumErrorLeve;  // No hay Error (Inicial)
      T     #NumErrorGrave;


      L     16;  // Long de la Estructura
      T     #LongBits;

      L     0;  // Offset de Los Bits
      T     #OffsetEmerg;
      L     2;
      T     #OffsetErrorGrave;
      L     4;
      T     #OffsetErrorLeve;

      L     15;  // Numero de Bits
      T     #MaxBitsGraves;
      L     95;
      T     #MaxBitsLeves;

      L     #Numero;
      T     #Zona;


///////////////////////////////////////////////////////////////////////////
// --- Comprobación del Numero de Dispositivo

      L     #Zona;
      L     0;
      <I;
      JC    Final;
      L     #Zona;
      L     "CTE_MaxDispositivos";
      >I;
      JC    Final;


///////////////////////////////////////////////////////////////////////////
// --- Calcular el Numero de Armario

      L     "CTE_OffsetCCPIF";
      L     100;
      *D;
      L     #Zona;
      +D;
      T     #Armario;

      JU    Mirar_EmergenciaGrave;  // Mirar a Emergencias Graves



NETWORK
TITLE = Codigo de Emegencia
Mirar_EmergenciaGrave:NOP   0;

///////////////////////////////////////////////////////////////////////////
// --- Preparar Puntero Inicial y Final

      L     #Zona;
      L     #LongBits;
      *D;
      L     #OffsetEmerg;
      +D;
      SLD   3;
      T     #P_Inicial;
      T     #P_Final;


///////////////////////////////////////////////////////////////////////////
// --- Recorrer el Arrray de Errores

Bucle_EmergenciaGrave:NOP   0;
      OPN   DB [#NumDB];  // Recorrer todos los Bits

      A     DBX [#P_Final];
      JC    Existe_EmergenciaGrave;  // Esta Activado este Bit

      L     #P_Final;
      L     #P_Inicial;
      -D;
      L     #MaxBitsGraves;
      ==I;
      JC    Final_EmergenciaGrave;  // Si ha recorrido todos los bits

      L     #P_Final;
      L     P#0.1;
      +D;
      T     #P_Final;
      JU    Bucle_EmergenciaGrave;  // Siguiente Bit


///////////////////////////////////////////////////////////////////////////
// --- Calcular el codigo

Existe_EmergenciaGrave:NOP   0;
      L     #P_Final;
      L     #P_Inicial;
      -D;
      L     1;  // Empieza 1 -> 16
      +D;
      T     #NumEmerg;  // Numero Bit Actrivado

      L     #NumEmerg;
      T     #ErrorFIFO;  // Codigo Final HMI


///////////////////////////////////////////////////////////////////////////
// ---      Escribir el Error
// ---      Preparar para Visualizar

      SET;
      S     #Emergencia;  // Activar Emergencia Grave

      L     #NumEmerg;  // Escribir Codigo
      T     #Codigo;

      L     #ErrorFIFO;
      T     "DB861_FIFO_Errores".ArmariosGraves[#Zona];

      JU    Final_EmergenciaGrave;  // Final


///////////////////////////////////////////////////////////////////////////
// --- No Hay EMergencia Grave

Final_EmergenciaGrave:NOP   0;  // No hay Graves
      JU    Mirar_ErrorGrave;  // Ir a Mirar los errores graves



NETWORK
TITLE = Codigo de Error de Grave
Mirar_ErrorGrave:NOP   0;

///////////////////////////////////////////////////////////////////////////
// --- Preparar Puntero Inicial y Final

      L     #Zona;
      L     #LongBits;
      *D;
      L     #OffsetErrorGrave;
      +D;
      SLD   3;
      T     #P_Inicial;
      T     #P_Final;


///////////////////////////////////////////////////////////////////////////
// --- Recorrer el Arrray de Errores

Bucle_ErrorGrave:NOP   0;
      OPN   DB [#NumDB];  // Recorrer todos los Bits
      A     DBX [#P_Final];
      JC    Existe_ErrorGrave;  // Esta Activado este Bit

      L     #P_Final;
      L     #P_Inicial;
      -D;
      L     #MaxBitsGraves;
      ==I;
      JC    Final_ErrorGrave;  // Si ha recorrido todos los bits

      L     #P_Final;
      L     P#0.1;
      +D;
      T     #P_Final;
      JU    Bucle_ErrorGrave;  // Siguiente Bit


///////////////////////////////////////////////////////////////////////////
// --- Calcular el Numero de Error

Existe_ErrorGrave:NOP   0;
      L     #P_Final;
      L     #P_Inicial;
      -D;
      L     100;  // Empieza 100 -> 199
      +D;
      T     #NumErrorGrave;  // Numero Bit Activado

      L     #NumErrorGrave;
      T     #ErrorFIFO;  // Codigo Final HMI

///////////////////////////////////////////////////////////////////////////
// ---      Escribir el Error
// ---      Preparar para Visualizar

      SET;
      S     #ErrorGrave;  // Activar Error Grave

      SET;
      A     #Emergencia;  // Escribir Codigo ?
      JC    NoActivarCodigo_ErrorGrave;

      L     #NumErrorGrave;
      T     #Codigo;

NoActivarCodigo_ErrorGrave:NOP   0;
      SET;
      A     #Emergencia;  // Guardar FIFO GRAVE ?
      JC    Final_ErrorGrave;

      L     #ErrorFIFO;
      T     "DB861_FIFO_Errores".ArmariosGraves[#Zona];

      JU    Final_ErrorGrave;  // Mirar Leves


///////////////////////////////////////////////////////////////////////////
// --- No Hay Error

Final_ErrorGrave:NOP   0;  // No hay Graves
      JU    MirarErrorLeve;  // Ir a Mirar los Leves



NETWORK
TITLE = Codigo de Error de Leves
///////////////////////////////////////////////////////////////////////////
// --- Preparar Puntero Inicial y Final

MirarErrorLeve:L     #Zona;
      L     #LongBits;
      *D;
      L     #OffsetErrorLeve;
      +D;
      SLD   3;
      T     #P_Inicial;
      T     #P_Final;  //nieves 28/08/25


///////////////////////////////////////////////////////////////////////////
// --- Recorrer el Arrray de Errores

Bucle_ErrorLeve:NOP   0;
      OPN   DB [#NumDB];  // Recorrer todos los Errores
      A     DBX [#P_Final];
      JC    Existe_ErrorLeve;  // Esta Activado este Bit

      L     #P_Final;
      L     #P_Inicial;
      -D;
      L     #MaxBitsLeves;
      ==I;
      JC    Final_ErrorLeve;  // Si ha recorrido todos los bits

      L     #P_Final;
      L     P#0.1;
      +D;
      T     #P_Final;
      JU    Bucle_ErrorLeve;  // Siguiente Bit


///////////////////////////////////////////////////////////////////////////
// --- Calcular el Numero de Error

Existe_ErrorLeve:NOP   0;
      L     #P_Final;
      L     #P_Inicial;
      -D;
      L     200;  //200 --> 299
      +D;
      T     #NumErrorLeve;  // Numero Bit Actrivado

      L     #NumErrorLeve;
      T     #ErrorFIFO;  // Codigo Final HMI


///////////////////////////////////////////////////////////////////////////
// ---      Escribir el Error
// ---      Preparar para Visualizar

      SET;
      S     #ErrorLeve;  // Activar Error Leve

      SET;
      A     #Emergencia;  // Escribir Codigo ?
      O     #ErrorGrave;
      JC    NoActivarCodigo_ErrorLeve;

      L     #NumErrorLeve;
      T     #Codigo;

NoActivarCodigo_ErrorLeve:NOP   0;
//      U     #Emergencia         // nieves comentado para que se activen tambien los errores leves aunque haya emergencia
//      SPB   Final

      L     #ErrorFIFO;
      T     "DB861_FIFO_Errores".ArmariosLeves[#Zona];

      JU    Final;  // No mirar más


///////////////////////////////////////////////////////////////////////////
// --- No Hay Error

Final_ErrorLeve:NOP   0;  // No hay Leves


///////////////////////////////////////////////////////////////////////////
// --- AUTO-REARME

      SET;
      R     #ErrorLeve;  // DesActivar Error Leve

      L     0;
      T     "DB861_FIFO_Errores".ArmariosLeves[#Zona];

      SET;
      A     #Emergencia;  // Borrado del Codigo ?
      O     #ErrorGrave;
      JC    Final;

      L     0;
      T     #Codigo;

      JU    Final;  // No hay mirar nadie más



NETWORK
TITLE = Finalizar
///////////////////////////////////////////////////////////////////////////
// --- Se acabo la Funcion

Final:NOP   0;



END_FUNCTION

FUNCTION "FC902_Decodifica_Selector" : Void   // FC902, LAD
TITLE = Digito de Selector
{ S7_Optimized_Access := 'FALSE' }
AUTHOR : GENERAL
NAME : 20150126
VERSION : 3.0
// stored: AutoNumber false, SetENOAutomatically false
   VAR_INPUT
      Bit_0 : Bool;
      Bit_1 : Bool;
      Bit_2 : Bool;
      Bit_3 : Bool;
   END_VAR
   VAR_OUTPUT
      Codigo : Word;
   END_VAR
BEGIN

REGION Network 1
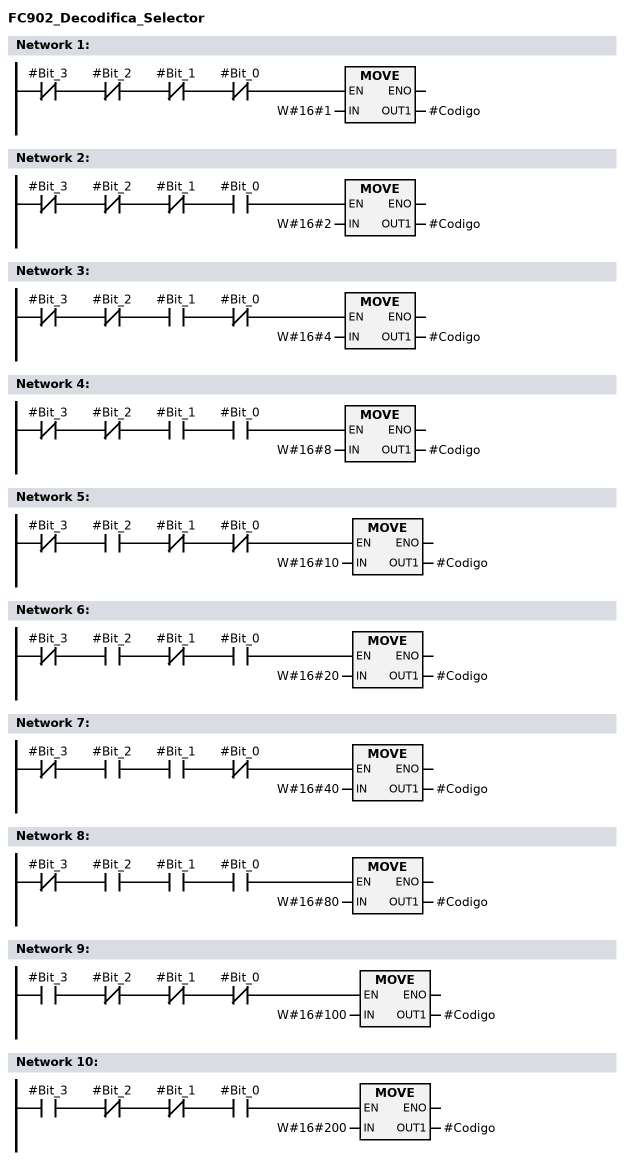
   RUNG wire#powerrail
      I_Contact( #Bit_3 )
      I_Contact( #Bit_2 )
      I_Contact( #Bit_1 )
      I_Contact( #Bit_0 )
      { S7_GenerateENO := "TRUE" } Move(in := W#16#1, out1 => #Codigo)
   END_RUNG
   // the same network as SCL:
   IF NOT #Bit_3 AND NOT #Bit_2 AND NOT #Bit_1 AND NOT #Bit_0 THEN #Codigo := W#16#1; END_IF;
END_REGION

REGION Network 2
   RUNG wire#powerrail
      I_Contact( #Bit_3 )
      I_Contact( #Bit_2 )
      I_Contact( #Bit_1 )
      Contact( #Bit_0 )
      { S7_GenerateENO := "TRUE" } Move(in := W#16#2, out1 => #Codigo)
   END_RUNG
   // the same network as SCL:
   IF NOT #Bit_3 AND NOT #Bit_2 AND NOT #Bit_1 AND #Bit_0 THEN #Codigo := W#16#2; END_IF;
END_REGION

REGION Network 3
   RUNG wire#powerrail
      I_Contact( #Bit_3 )
      I_Contact( #Bit_2 )
      Contact( #Bit_1 )
      I_Contact( #Bit_0 )
      { S7_GenerateENO := "TRUE" } Move(in := W#16#4, out1 => #Codigo)
   END_RUNG
   // the same network as SCL:
   IF NOT #Bit_3 AND NOT #Bit_2 AND #Bit_1 AND NOT #Bit_0 THEN #Codigo := W#16#4; END_IF;
END_REGION

REGION Network 4
   RUNG wire#powerrail
      I_Contact( #Bit_3 )
      I_Contact( #Bit_2 )
      Contact( #Bit_1 )
      Contact( #Bit_0 )
      { S7_GenerateENO := "TRUE" } Move(in := W#16#8, out1 => #Codigo)
   END_RUNG
   // the same network as SCL:
   IF NOT #Bit_3 AND NOT #Bit_2 AND #Bit_1 AND #Bit_0 THEN #Codigo := W#16#8; END_IF;
END_REGION

REGION Network 5
   RUNG wire#powerrail
      I_Contact( #Bit_3 )
      Contact( #Bit_2 )
      I_Contact( #Bit_1 )
      I_Contact( #Bit_0 )
      { S7_GenerateENO := "TRUE" } Move(in := W#16#10, out1 => #Codigo)
   END_RUNG
   // the same network as SCL:
   IF NOT #Bit_3 AND #Bit_2 AND NOT #Bit_1 AND NOT #Bit_0 THEN #Codigo := W#16#10; END_IF;
END_REGION

REGION Network 6
   RUNG wire#powerrail
      I_Contact( #Bit_3 )
      Contact( #Bit_2 )
      I_Contact( #Bit_1 )
      Contact( #Bit_0 )
      { S7_GenerateENO := "TRUE" } Move(in := W#16#20, out1 => #Codigo)
   END_RUNG
   // the same network as SCL:
   IF NOT #Bit_3 AND #Bit_2 AND NOT #Bit_1 AND #Bit_0 THEN #Codigo := W#16#20; END_IF;
END_REGION

REGION Network 7
   RUNG wire#powerrail
      I_Contact( #Bit_3 )
      Contact( #Bit_2 )
      Contact( #Bit_1 )
      I_Contact( #Bit_0 )
      { S7_GenerateENO := "TRUE" } Move(in := W#16#40, out1 => #Codigo)
   END_RUNG
   // the same network as SCL:
   IF NOT #Bit_3 AND #Bit_2 AND #Bit_1 AND NOT #Bit_0 THEN #Codigo := W#16#40; END_IF;
END_REGION

REGION Network 8
   RUNG wire#powerrail
      I_Contact( #Bit_3 )
      Contact( #Bit_2 )
      Contact( #Bit_1 )
      Contact( #Bit_0 )
      { S7_GenerateENO := "TRUE" } Move(in := W#16#80, out1 => #Codigo)
   END_RUNG
   // the same network as SCL:
   IF NOT #Bit_3 AND #Bit_2 AND #Bit_1 AND #Bit_0 THEN #Codigo := W#16#80; END_IF;
END_REGION

REGION Network 9
   RUNG wire#powerrail
      Contact( #Bit_3 )
      I_Contact( #Bit_2 )
      I_Contact( #Bit_1 )
      I_Contact( #Bit_0 )
      { S7_GenerateENO := "TRUE" } Move(in := W#16#100, out1 => #Codigo)
   END_RUNG
   // the same network as SCL:
   IF #Bit_3 AND NOT #Bit_2 AND NOT #Bit_1 AND NOT #Bit_0 THEN #Codigo := W#16#100; END_IF;
END_REGION

REGION Network 10
   RUNG wire#powerrail
      Contact( #Bit_3 )
      I_Contact( #Bit_2 )
      I_Contact( #Bit_1 )
      Contact( #Bit_0 )
      { S7_GenerateENO := "TRUE" } Move(in := W#16#200, out1 => #Codigo)
   END_RUNG
   // the same network as SCL:
   IF #Bit_3 AND NOT #Bit_2 AND NOT #Bit_1 AND #Bit_0 THEN #Codigo := W#16#200; END_IF;
END_REGION
END_FUNCTION

FUNCTION "FC910_CNT_pulsos_UHS" : Void   // FC910, LAD
{ S7_Optimized_Access := 'FALSE' }
AUTHOR : GENERAL
NAME : 20130301
VERSION : 3.0
// stored: AutoNumber false, SetENOAutomatically false
   VAR_INPUT
      CUENTA_UP : Bool;
      RESET : Bool;
      Valor_Cuenta : UDInt;
   END_VAR
   VAR_OUTPUT
      Cuenta_OK : Bool;
   END_VAR
   VAR_IN_OUT
      Valor_Actual : UDInt;
   END_VAR
   VAR_TEMP
      TEMP_Cuenta_OK : Bool;
   END_VAR
BEGIN

REGION Network 1
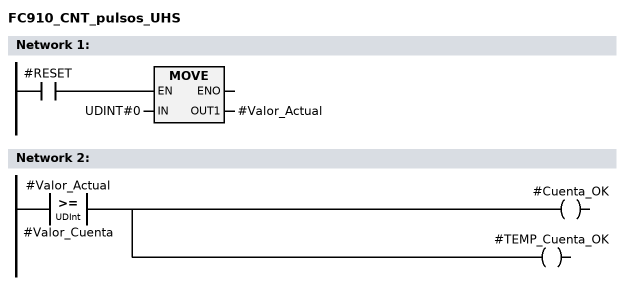
   RUNG wire#powerrail
      Contact( #RESET )
      { S7_GenerateENO := "TRUE" } Move(in := UDINT#0, out1 => #Valor_Actual)
   END_RUNG
   // the same network as SCL:
   IF #RESET THEN #Valor_Actual := UDINT#0; END_IF;
END_REGION

REGION Network 2
   RUNG wire#powerrail
      { S7_Templates := "SrcType := UDInt" } GE_Contact(in1 := #Valor_Actual, in2 := #Valor_Cuenta)
      wire#w1
      Coil( #Cuenta_OK )
   END_RUNG
   RUNG wire#w1
      Coil( #TEMP_Cuenta_OK )
   END_RUNG
   // the same network as SCL:
   #Cuenta_OK := #Valor_Actual >= #Valor_Cuenta;
   #TEMP_Cuenta_OK := #Cuenta_OK;
END_REGION

NETWORK
TITLE = 
      A     #CUENTA_UP;
      AN    #TEMP_Cuenta_OK;
      JNB   _002;
      L     #Valor_Actual;
      L     1;
      +D;
      T     #Valor_Actual;
_002: NOP   0;
END_FUNCTION

FUNCTION "FC920_Registro_Flujos" : Void   // FC920, LAD
TITLE = FC920_Registro_Flujos
{ S7_Optimized_Access := 'FALSE' }
// FC920 Registro Flujos
// stored: AutoNumber false, SetENOAutomatically false
   VAR_INPUT
      Numero_mesa : Int;
   END_VAR
   VAR_TEMP
      cambia_registro : Bool;
      cero : Int;
      retval : Int;
      ROD_CAD : DInt;
      Registro_vacio : Struct
         registro : Array[1..10] of "Registro";
      END_STRUCT;
   END_VAR
   VAR_TEMP   // added for the SCL form of the ladder/FBD networks
      _w1 : Bool;
      _w2 : Bool;
      _w3 : Bool;
      _w4 : Bool;
   END_VAR
BEGIN

REGION Network 1: Inicializacion y cambio de registro registro para poder hacer varios registros
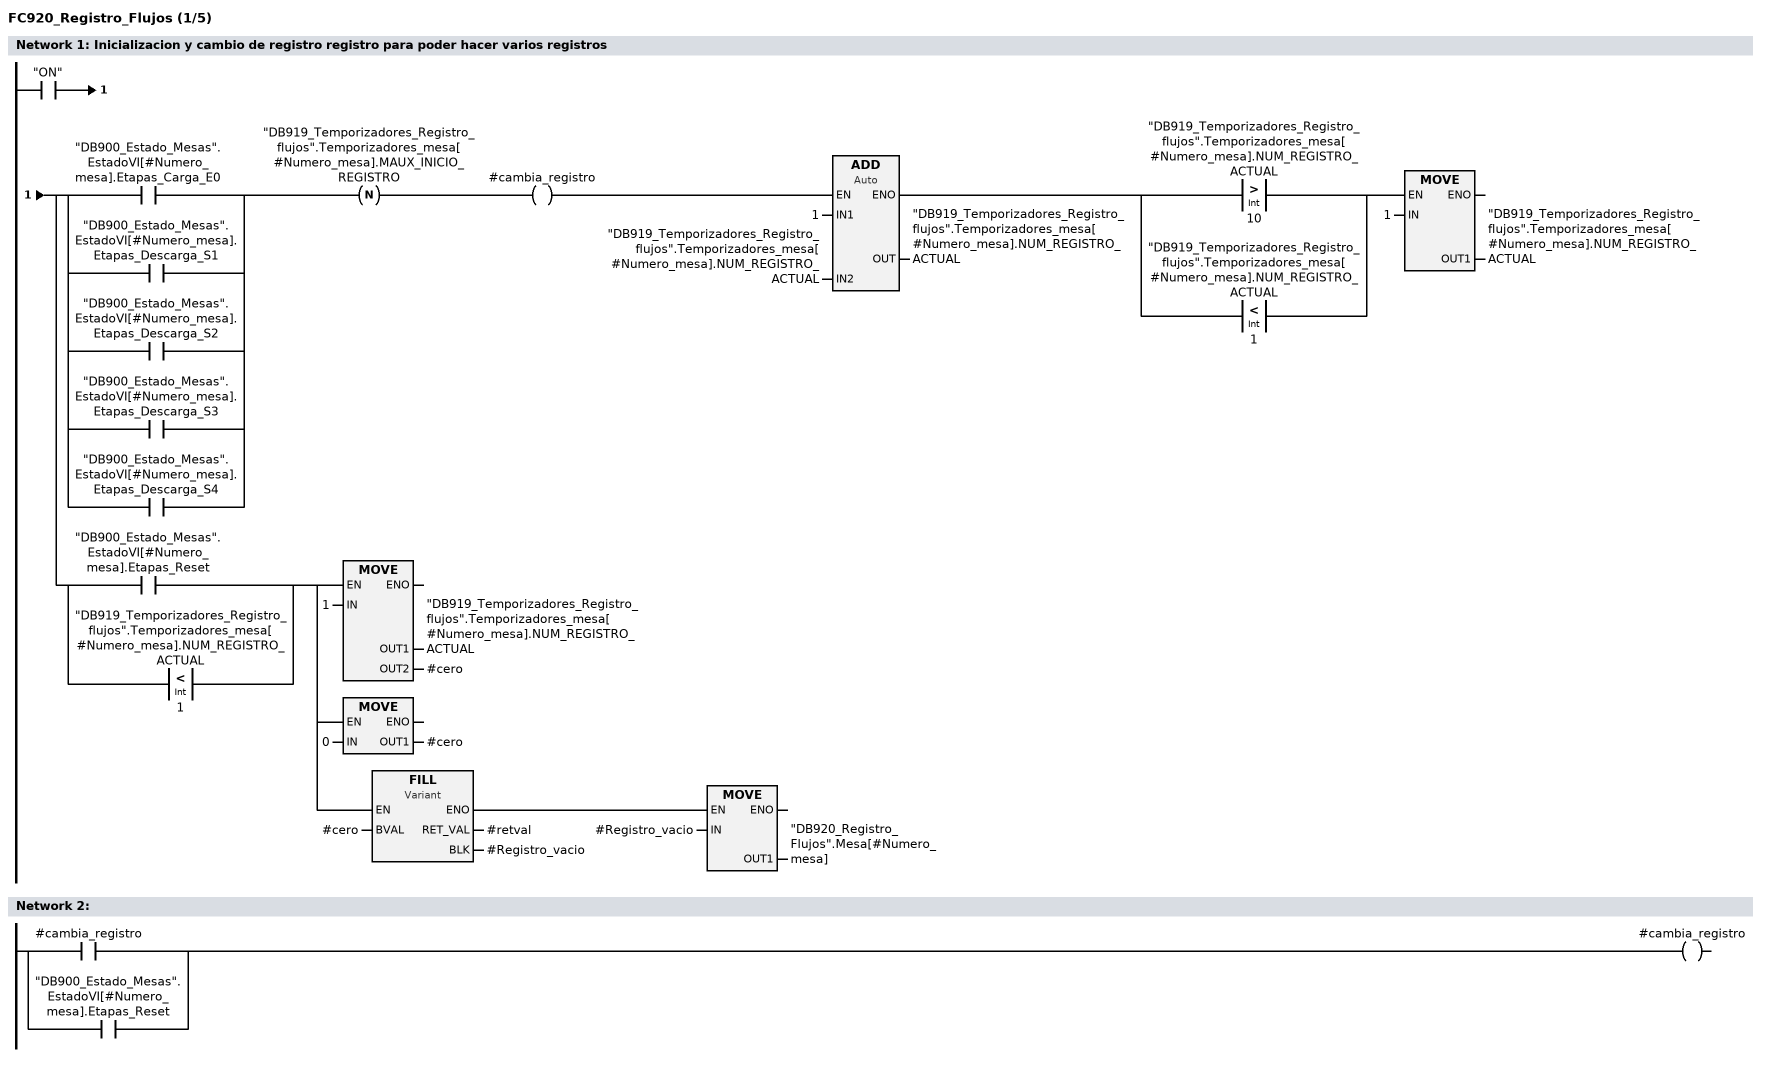
   RUNG wire#powerrail
      Contact( "ON" )
      wire#w1
      Contact( "DB900_Estado_Mesas".EstadoVI[#Numero_mesa].Etapas_Carga_E0 )
      wire#w2
      N_Trig( "DB919_Temporizadores_Registro_flujos".Temporizadores_mesa[#Numero_mesa].MAUX_INICIO_REGISTRO )
      Coil( #cambia_registro )
      Add(in1 := 1, in2 := "DB919_Temporizadores_Registro_flujos".Temporizadores_mesa[#Numero_mesa].NUM_REGISTRO_ACTUAL, out => "DB919_Temporizadores_Registro_flujos".Temporizadores_mesa[#Numero_mesa].NUM_REGISTRO_ACTUAL)
      wire#w3
      { S7_Templates := "SrcType := Int" } GT_Contact(in1 := "DB919_Temporizadores_Registro_flujos".Temporizadores_mesa[#Numero_mesa].NUM_REGISTRO_ACTUAL, in2 := 10)
      wire#w4
      Move(in := 1, out1 => "DB919_Temporizadores_Registro_flujos".Temporizadores_mesa[#Numero_mesa].NUM_REGISTRO_ACTUAL)
   END_RUNG
   RUNG wire#w1
      Contact( "DB900_Estado_Mesas".EstadoVI[#Numero_mesa].Etapas_Descarga_S1 )
   END_RUNG wire#w2
   RUNG wire#w1
      Contact( "DB900_Estado_Mesas".EstadoVI[#Numero_mesa].Etapas_Descarga_S2 )
   END_RUNG wire#w2
   RUNG wire#w1
      Contact( "DB900_Estado_Mesas".EstadoVI[#Numero_mesa].Etapas_Descarga_S3 )
   END_RUNG wire#w2
   RUNG wire#w1
      Contact( "DB900_Estado_Mesas".EstadoVI[#Numero_mesa].Etapas_Descarga_S4 )
   END_RUNG wire#w2
   RUNG wire#w3
      { S7_Templates := "SrcType := Int" } LT_Contact(in1 := "DB919_Temporizadores_Registro_flujos".Temporizadores_mesa[#Numero_mesa].NUM_REGISTRO_ACTUAL, in2 := 1)
   END_RUNG wire#w4
   RUNG wire#w1
      Contact( "DB900_Estado_Mesas".EstadoVI[#Numero_mesa].Etapas_Reset )
      wire#w5
      Move(in := 1, out1 => "DB919_Temporizadores_Registro_flujos".Temporizadores_mesa[#Numero_mesa].NUM_REGISTRO_ACTUAL, out2 => #cero)
   END_RUNG
   RUNG wire#w1
      { S7_Templates := "SrcType := Int" } LT_Contact(in1 := "DB919_Temporizadores_Registro_flujos".Temporizadores_mesa[#Numero_mesa].NUM_REGISTRO_ACTUAL, in2 := 1)
   END_RUNG wire#w5
   RUNG wire#w5
      Move(in := 0, out1 => #cero)
   END_RUNG
   RUNG wire#w5
      { S7_Templates := "ptr_type := Variant" } FILL(BVAL := #cero, RET_VAL => #retval, BLK => #Registro_vacio)
      Move(in := #Registro_vacio, out1 => "DB920_Registro_Flujos".Mesa[#Numero_mesa])
   END_RUNG
   // the same network as SCL:
   #_w1 := "ON" AND ("DB900_Estado_Mesas".EstadoVI[#Numero_mesa].Etapas_Carga_E0 OR "DB900_Estado_Mesas".EstadoVI[#Numero_mesa].Etapas_Descarga_S1 OR "DB900_Estado_Mesas".EstadoVI[#Numero_mesa].Etapas_Descarga_S2 OR "DB900_Estado_Mesas".EstadoVI[#Numero_mesa].Etapas_Descarga_S3 OR "DB900_Estado_Mesas".EstadoVI[#Numero_mesa].Etapas_Descarga_S4);
   #_w2 := NOT #_w1 AND "DB919_Temporizadores_Registro_flujos".Temporizadores_mesa[#Numero_mesa].MAUX_INICIO_REGISTRO;   // falling edge
   "DB919_Temporizadores_Registro_flujos".Temporizadores_mesa[#Numero_mesa].MAUX_INICIO_REGISTRO := #_w1;
   #cambia_registro := #_w2;
   IF #_w2 THEN
       "DB919_Temporizadores_Registro_flujos".Temporizadores_mesa[#Numero_mesa].NUM_REGISTRO_ACTUAL := 1 + "DB919_Temporizadores_Registro_flujos".Temporizadores_mesa[#Numero_mesa].NUM_REGISTRO_ACTUAL;
   END_IF;
   IF #_w2 AND (("DB919_Temporizadores_Registro_flujos".Temporizadores_mesa[#Numero_mesa].NUM_REGISTRO_ACTUAL > 10) OR ("DB919_Temporizadores_Registro_flujos".Temporizadores_mesa[#Numero_mesa].NUM_REGISTRO_ACTUAL < 1)) THEN
       "DB919_Temporizadores_Registro_flujos".Temporizadores_mesa[#Numero_mesa].NUM_REGISTRO_ACTUAL := 1;
   END_IF;
   #_w3 := "ON" AND ("DB900_Estado_Mesas".EstadoVI[#Numero_mesa].Etapas_Reset OR ("DB919_Temporizadores_Registro_flujos".Temporizadores_mesa[#Numero_mesa].NUM_REGISTRO_ACTUAL < 1));
   IF #_w3 THEN
       "DB919_Temporizadores_Registro_flujos".Temporizadores_mesa[#Numero_mesa].NUM_REGISTRO_ACTUAL := 1;
       #cero := 1;
       #cero := 0;
   END_IF;
   #retval := FILL(EN := #_w3, BVAL := #cero, BLK => #Registro_vacio, ENO => #_w4);
   IF #_w4 THEN "DB920_Registro_Flujos".Mesa[#Numero_mesa] := #Registro_vacio; END_IF;
END_REGION

REGION Network 2
   RUNG wire#powerrail
      Contact( #cambia_registro )
      wire#w1
      Coil( #cambia_registro )
   END_RUNG
   RUNG wire#powerrail
      Contact( "DB900_Estado_Mesas".EstadoVI[#Numero_mesa].Etapas_Reset )
   END_RUNG wire#w1
   // the same network as SCL:
   #cambia_registro := #cambia_registro OR "DB900_Estado_Mesas".EstadoVI[#Numero_mesa].Etapas_Reset;
END_REGION

REGION Network 3: Temporizador Etapas de Carga
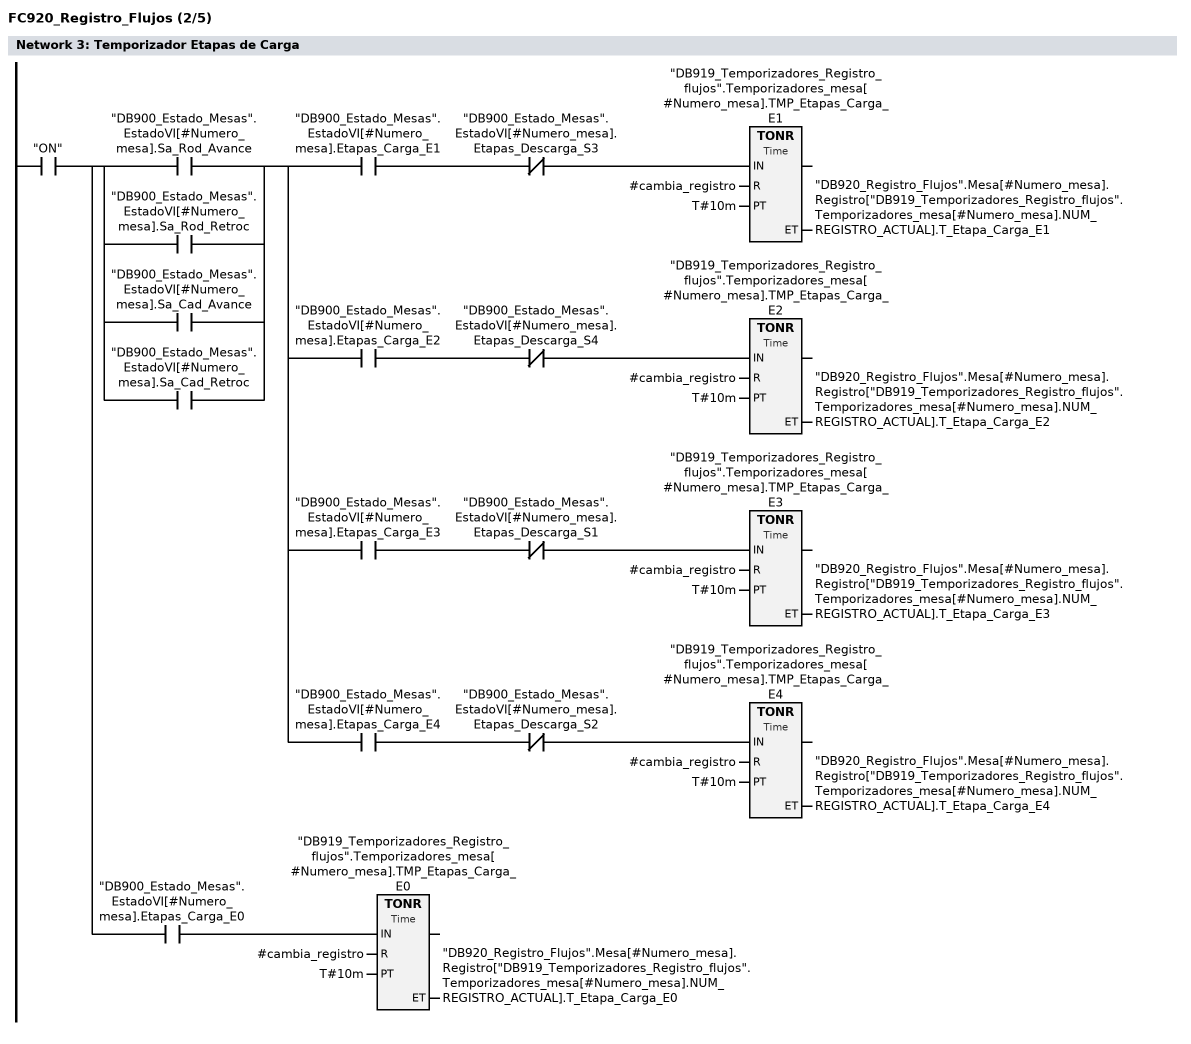
   RUNG wire#powerrail
      Contact( "ON" )
      wire#w1
      Contact( "DB900_Estado_Mesas".EstadoVI[#Numero_mesa].Sa_Rod_Avance )
      wire#w2
      Contact( "DB900_Estado_Mesas".EstadoVI[#Numero_mesa].Etapas_Carga_E1 )
      I_Contact( "DB900_Estado_Mesas".EstadoVI[#Numero_mesa].Etapas_Descarga_S3 )
      { S7_Templates := "time_type := Time" } "DB919_Temporizadores_Registro_flujos".Temporizadores_mesa[#Numero_mesa].TMP_Etapas_Carga_E1.TONR(r := #cambia_registro, pt := T#10m, et => "DB920_Registro_Flujos".Mesa[#Numero_mesa].Registro["DB919_Temporizadores_Registro_flujos".Temporizadores_mesa[#Numero_mesa].NUM_REGISTRO_ACTUAL].T_Etapa_Carga_E1)
   END_RUNG
   RUNG wire#w1
      Contact( "DB900_Estado_Mesas".EstadoVI[#Numero_mesa].Sa_Rod_Retroc )
   END_RUNG wire#w2
   RUNG wire#w1
      Contact( "DB900_Estado_Mesas".EstadoVI[#Numero_mesa].Sa_Cad_Avance )
   END_RUNG wire#w2
   RUNG wire#w1
      Contact( "DB900_Estado_Mesas".EstadoVI[#Numero_mesa].Sa_Cad_Retroc )
   END_RUNG wire#w2
   RUNG wire#w2
      Contact( "DB900_Estado_Mesas".EstadoVI[#Numero_mesa].Etapas_Carga_E2 )
      I_Contact( "DB900_Estado_Mesas".EstadoVI[#Numero_mesa].Etapas_Descarga_S4 )
      { S7_Templates := "time_type := Time" } "DB919_Temporizadores_Registro_flujos".Temporizadores_mesa[#Numero_mesa].TMP_Etapas_Carga_E2.TONR(r := #cambia_registro, pt := T#10m, et => "DB920_Registro_Flujos".Mesa[#Numero_mesa].Registro["DB919_Temporizadores_Registro_flujos".Temporizadores_mesa[#Numero_mesa].NUM_REGISTRO_ACTUAL].T_Etapa_Carga_E2)
   END_RUNG
   RUNG wire#w2
      Contact( "DB900_Estado_Mesas".EstadoVI[#Numero_mesa].Etapas_Carga_E3 )
      I_Contact( "DB900_Estado_Mesas".EstadoVI[#Numero_mesa].Etapas_Descarga_S1 )
      { S7_Templates := "time_type := Time" } "DB919_Temporizadores_Registro_flujos".Temporizadores_mesa[#Numero_mesa].TMP_Etapas_Carga_E3.TONR(r := #cambia_registro, pt := T#10m, et => "DB920_Registro_Flujos".Mesa[#Numero_mesa].Registro["DB919_Temporizadores_Registro_flujos".Temporizadores_mesa[#Numero_mesa].NUM_REGISTRO_ACTUAL].T_Etapa_Carga_E3)
   END_RUNG
   RUNG wire#w2
      Contact( "DB900_Estado_Mesas".EstadoVI[#Numero_mesa].Etapas_Carga_E4 )
      I_Contact( "DB900_Estado_Mesas".EstadoVI[#Numero_mesa].Etapas_Descarga_S2 )
      { S7_Templates := "time_type := Time" } "DB919_Temporizadores_Registro_flujos".Temporizadores_mesa[#Numero_mesa].TMP_Etapas_Carga_E4.TONR(r := #cambia_registro, pt := T#10m, et => "DB920_Registro_Flujos".Mesa[#Numero_mesa].Registro["DB919_Temporizadores_Registro_flujos".Temporizadores_mesa[#Numero_mesa].NUM_REGISTRO_ACTUAL].T_Etapa_Carga_E4)
   END_RUNG
   RUNG wire#w1
      Contact( "DB900_Estado_Mesas".EstadoVI[#Numero_mesa].Etapas_Carga_E0 )
      { S7_Templates := "time_type := Time" } "DB919_Temporizadores_Registro_flujos".Temporizadores_mesa[#Numero_mesa].TMP_Etapas_Carga_E0.TONR(r := #cambia_registro, pt := T#10m, et => "DB920_Registro_Flujos".Mesa[#Numero_mesa].Registro["DB919_Temporizadores_Registro_flujos".Temporizadores_mesa[#Numero_mesa].NUM_REGISTRO_ACTUAL].T_Etapa_Carga_E0)
   END_RUNG
   // the same network as SCL:
   #_w1 := "ON" AND ("DB900_Estado_Mesas".EstadoVI[#Numero_mesa].Sa_Rod_Avance OR "DB900_Estado_Mesas".EstadoVI[#Numero_mesa].Sa_Rod_Retroc OR "DB900_Estado_Mesas".EstadoVI[#Numero_mesa].Sa_Cad_Avance OR "DB900_Estado_Mesas".EstadoVI[#Numero_mesa].Sa_Cad_Retroc);
   "DB919_Temporizadores_Registro_flujos".Temporizadores_mesa[#Numero_mesa].TMP_Etapas_Carga_E1.TONR(IN := #_w1 AND "DB900_Estado_Mesas".EstadoVI[#Numero_mesa].Etapas_Carga_E1 AND NOT "DB900_Estado_Mesas".EstadoVI[#Numero_mesa].Etapas_Descarga_S3,
                           R := #cambia_registro,
                           PT := T#10m,
                           ET => "DB920_Registro_Flujos".Mesa[#Numero_mesa].Registro["DB919_Temporizadores_Registro_flujos".Temporizadores_mesa[#Numero_mesa].NUM_REGISTRO_ACTUAL].T_Etapa_Carga_E1);
   "DB919_Temporizadores_Registro_flujos".Temporizadores_mesa[#Numero_mesa].TMP_Etapas_Carga_E2.TONR(IN := #_w1 AND "DB900_Estado_Mesas".EstadoVI[#Numero_mesa].Etapas_Carga_E2 AND NOT "DB900_Estado_Mesas".EstadoVI[#Numero_mesa].Etapas_Descarga_S4,
                           R := #cambia_registro,
                           PT := T#10m,
                           ET => "DB920_Registro_Flujos".Mesa[#Numero_mesa].Registro["DB919_Temporizadores_Registro_flujos".Temporizadores_mesa[#Numero_mesa].NUM_REGISTRO_ACTUAL].T_Etapa_Carga_E2);
   "DB919_Temporizadores_Registro_flujos".Temporizadores_mesa[#Numero_mesa].TMP_Etapas_Carga_E3.TONR(IN := #_w1 AND "DB900_Estado_Mesas".EstadoVI[#Numero_mesa].Etapas_Carga_E3 AND NOT "DB900_Estado_Mesas".EstadoVI[#Numero_mesa].Etapas_Descarga_S1,
                           R := #cambia_registro,
                           PT := T#10m,
                           ET => "DB920_Registro_Flujos".Mesa[#Numero_mesa].Registro["DB919_Temporizadores_Registro_flujos".Temporizadores_mesa[#Numero_mesa].NUM_REGISTRO_ACTUAL].T_Etapa_Carga_E3);
   "DB919_Temporizadores_Registro_flujos".Temporizadores_mesa[#Numero_mesa].TMP_Etapas_Carga_E4.TONR(IN := #_w1 AND "DB900_Estado_Mesas".EstadoVI[#Numero_mesa].Etapas_Carga_E4 AND NOT "DB900_Estado_Mesas".EstadoVI[#Numero_mesa].Etapas_Descarga_S2,
                           R := #cambia_registro,
                           PT := T#10m,
                           ET => "DB920_Registro_Flujos".Mesa[#Numero_mesa].Registro["DB919_Temporizadores_Registro_flujos".Temporizadores_mesa[#Numero_mesa].NUM_REGISTRO_ACTUAL].T_Etapa_Carga_E4);
   "DB919_Temporizadores_Registro_flujos".Temporizadores_mesa[#Numero_mesa].TMP_Etapas_Carga_E0.TONR(IN := "ON" AND "DB900_Estado_Mesas".EstadoVI[#Numero_mesa].Etapas_Carga_E0,
                           R := #cambia_registro,
                           PT := T#10m,
                           ET => "DB920_Registro_Flujos".Mesa[#Numero_mesa].Registro["DB919_Temporizadores_Registro_flujos".Temporizadores_mesa[#Numero_mesa].NUM_REGISTRO_ACTUAL].T_Etapa_Carga_E0);
END_REGION

REGION Network 4: Temporizador Etapas de Descarga
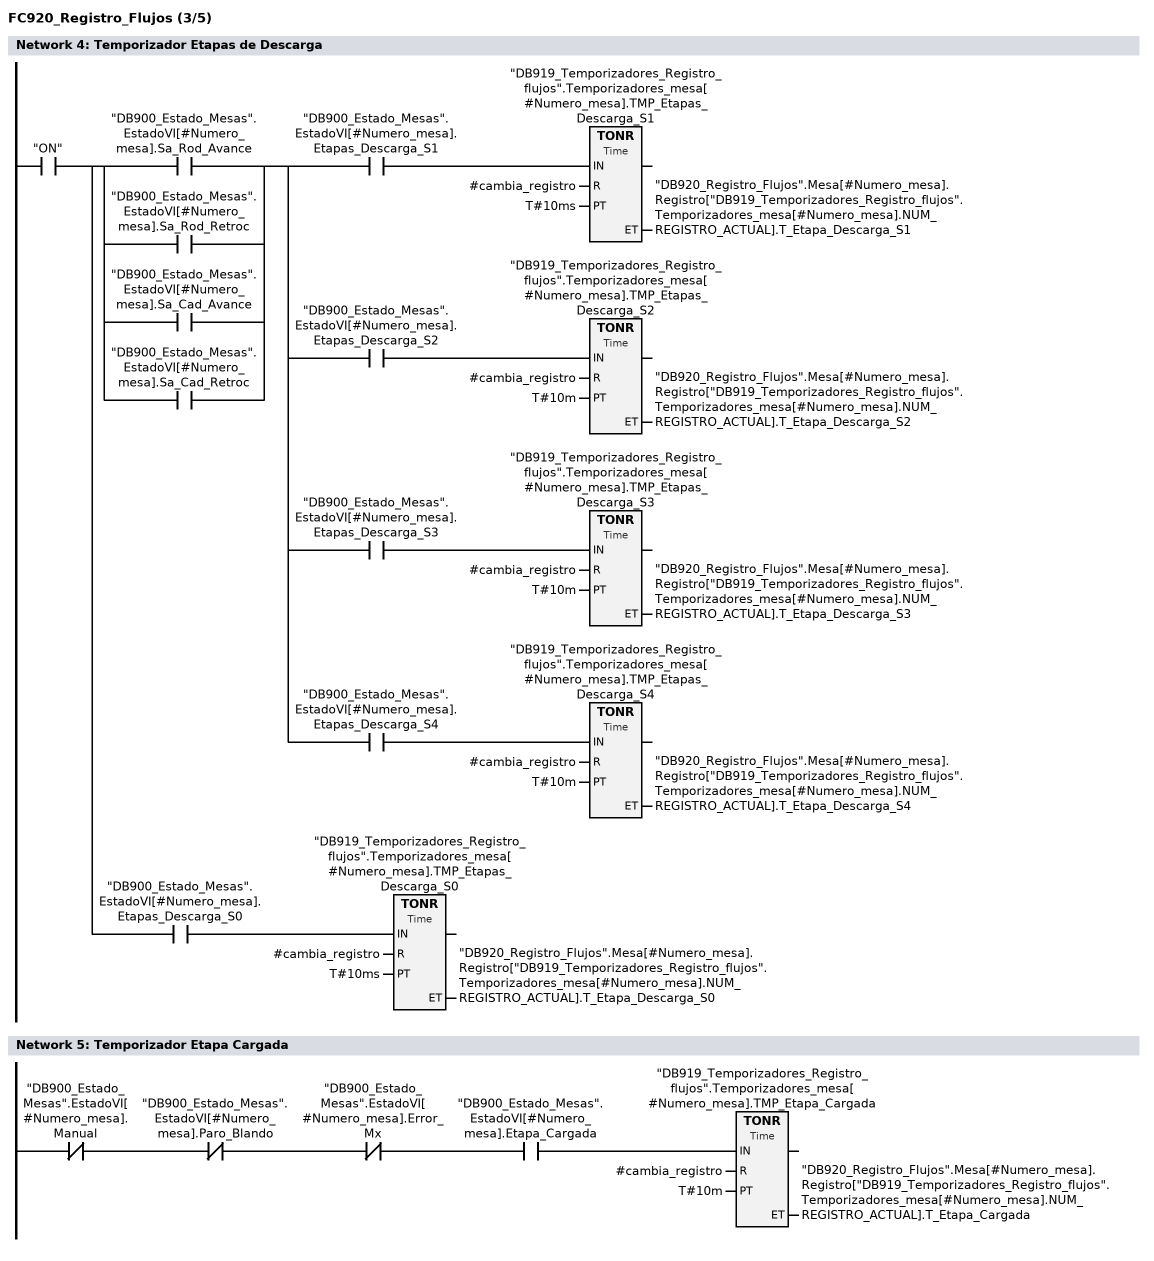
   RUNG wire#powerrail
      Contact( "ON" )
      wire#w1
      Contact( "DB900_Estado_Mesas".EstadoVI[#Numero_mesa].Sa_Rod_Avance )
      wire#w2
      Contact( "DB900_Estado_Mesas".EstadoVI[#Numero_mesa].Etapas_Descarga_S1 )
      { S7_Templates := "time_type := Time" } "DB919_Temporizadores_Registro_flujos".Temporizadores_mesa[#Numero_mesa].TMP_Etapas_Descarga_S1.TONR(r := #cambia_registro, pt := T#10ms, et => "DB920_Registro_Flujos".Mesa[#Numero_mesa].Registro["DB919_Temporizadores_Registro_flujos".Temporizadores_mesa[#Numero_mesa].NUM_REGISTRO_ACTUAL].T_Etapa_Descarga_S1)
   END_RUNG
   RUNG wire#w1
      Contact( "DB900_Estado_Mesas".EstadoVI[#Numero_mesa].Sa_Rod_Retroc )
   END_RUNG wire#w2
   RUNG wire#w1
      Contact( "DB900_Estado_Mesas".EstadoVI[#Numero_mesa].Sa_Cad_Avance )
   END_RUNG wire#w2
   RUNG wire#w1
      Contact( "DB900_Estado_Mesas".EstadoVI[#Numero_mesa].Sa_Cad_Retroc )
   END_RUNG wire#w2
   RUNG wire#w2
      Contact( "DB900_Estado_Mesas".EstadoVI[#Numero_mesa].Etapas_Descarga_S2 )
      { S7_Templates := "time_type := Time" } "DB919_Temporizadores_Registro_flujos".Temporizadores_mesa[#Numero_mesa].TMP_Etapas_Descarga_S2.TONR(r := #cambia_registro, pt := T#10m, et => "DB920_Registro_Flujos".Mesa[#Numero_mesa].Registro["DB919_Temporizadores_Registro_flujos".Temporizadores_mesa[#Numero_mesa].NUM_REGISTRO_ACTUAL].T_Etapa_Descarga_S2)
   END_RUNG
   RUNG wire#w2
      Contact( "DB900_Estado_Mesas".EstadoVI[#Numero_mesa].Etapas_Descarga_S3 )
      { S7_Templates := "time_type := Time" } "DB919_Temporizadores_Registro_flujos".Temporizadores_mesa[#Numero_mesa].TMP_Etapas_Descarga_S3.TONR(r := #cambia_registro, pt := T#10m, et => "DB920_Registro_Flujos".Mesa[#Numero_mesa].Registro["DB919_Temporizadores_Registro_flujos".Temporizadores_mesa[#Numero_mesa].NUM_REGISTRO_ACTUAL].T_Etapa_Descarga_S3)
   END_RUNG
   RUNG wire#w2
      Contact( "DB900_Estado_Mesas".EstadoVI[#Numero_mesa].Etapas_Descarga_S4 )
      { S7_Templates := "time_type := Time" } "DB919_Temporizadores_Registro_flujos".Temporizadores_mesa[#Numero_mesa].TMP_Etapas_Descarga_S4.TONR(r := #cambia_registro, pt := T#10m, et => "DB920_Registro_Flujos".Mesa[#Numero_mesa].Registro["DB919_Temporizadores_Registro_flujos".Temporizadores_mesa[#Numero_mesa].NUM_REGISTRO_ACTUAL].T_Etapa_Descarga_S4)
   END_RUNG
   RUNG wire#w1
      Contact( "DB900_Estado_Mesas".EstadoVI[#Numero_mesa].Etapas_Descarga_S0 )
      { S7_Templates := "time_type := Time" } "DB919_Temporizadores_Registro_flujos".Temporizadores_mesa[#Numero_mesa].TMP_Etapas_Descarga_S0.TONR(r := #cambia_registro, pt := T#10ms, et => "DB920_Registro_Flujos".Mesa[#Numero_mesa].Registro["DB919_Temporizadores_Registro_flujos".Temporizadores_mesa[#Numero_mesa].NUM_REGISTRO_ACTUAL].T_Etapa_Descarga_S0)
   END_RUNG
   // the same network as SCL:
   #_w1 := "ON" AND ("DB900_Estado_Mesas".EstadoVI[#Numero_mesa].Sa_Rod_Avance OR "DB900_Estado_Mesas".EstadoVI[#Numero_mesa].Sa_Rod_Retroc OR "DB900_Estado_Mesas".EstadoVI[#Numero_mesa].Sa_Cad_Avance OR "DB900_Estado_Mesas".EstadoVI[#Numero_mesa].Sa_Cad_Retroc);
   "DB919_Temporizadores_Registro_flujos".Temporizadores_mesa[#Numero_mesa].TMP_Etapas_Descarga_S1.TONR(IN := #_w1 AND "DB900_Estado_Mesas".EstadoVI[#Numero_mesa].Etapas_Descarga_S1,
                           R := #cambia_registro,
                           PT := T#10ms,
                           ET => "DB920_Registro_Flujos".Mesa[#Numero_mesa].Registro["DB919_Temporizadores_Registro_flujos".Temporizadores_mesa[#Numero_mesa].NUM_REGISTRO_ACTUAL].T_Etapa_Descarga_S1);
   "DB919_Temporizadores_Registro_flujos".Temporizadores_mesa[#Numero_mesa].TMP_Etapas_Descarga_S2.TONR(IN := #_w1 AND "DB900_Estado_Mesas".EstadoVI[#Numero_mesa].Etapas_Descarga_S2,
                           R := #cambia_registro,
                           PT := T#10m,
                           ET => "DB920_Registro_Flujos".Mesa[#Numero_mesa].Registro["DB919_Temporizadores_Registro_flujos".Temporizadores_mesa[#Numero_mesa].NUM_REGISTRO_ACTUAL].T_Etapa_Descarga_S2);
   "DB919_Temporizadores_Registro_flujos".Temporizadores_mesa[#Numero_mesa].TMP_Etapas_Descarga_S3.TONR(IN := #_w1 AND "DB900_Estado_Mesas".EstadoVI[#Numero_mesa].Etapas_Descarga_S3,
                           R := #cambia_registro,
                           PT := T#10m,
                           ET => "DB920_Registro_Flujos".Mesa[#Numero_mesa].Registro["DB919_Temporizadores_Registro_flujos".Temporizadores_mesa[#Numero_mesa].NUM_REGISTRO_ACTUAL].T_Etapa_Descarga_S3);
   "DB919_Temporizadores_Registro_flujos".Temporizadores_mesa[#Numero_mesa].TMP_Etapas_Descarga_S4.TONR(IN := #_w1 AND "DB900_Estado_Mesas".EstadoVI[#Numero_mesa].Etapas_Descarga_S4,
                           R := #cambia_registro,
                           PT := T#10m,
                           ET => "DB920_Registro_Flujos".Mesa[#Numero_mesa].Registro["DB919_Temporizadores_Registro_flujos".Temporizadores_mesa[#Numero_mesa].NUM_REGISTRO_ACTUAL].T_Etapa_Descarga_S4);
   "DB919_Temporizadores_Registro_flujos".Temporizadores_mesa[#Numero_mesa].TMP_Etapas_Descarga_S0.TONR(IN := "ON" AND "DB900_Estado_Mesas".EstadoVI[#Numero_mesa].Etapas_Descarga_S0,
                           R := #cambia_registro,
                           PT := T#10ms,
                           ET => "DB920_Registro_Flujos".Mesa[#Numero_mesa].Registro["DB919_Temporizadores_Registro_flujos".Temporizadores_mesa[#Numero_mesa].NUM_REGISTRO_ACTUAL].T_Etapa_Descarga_S0);
END_REGION

REGION Network 5: Temporizador Etapa Cargada
   RUNG wire#powerrail
      I_Contact( "DB900_Estado_Mesas".EstadoVI[#Numero_mesa].Manual )
      I_Contact( "DB900_Estado_Mesas".EstadoVI[#Numero_mesa].Paro_Blando )
      I_Contact( "DB900_Estado_Mesas".EstadoVI[#Numero_mesa].Error_Mx )
      Contact( "DB900_Estado_Mesas".EstadoVI[#Numero_mesa].Etapa_Cargada )
      { S7_Templates := "time_type := Time" } "DB919_Temporizadores_Registro_flujos".Temporizadores_mesa[#Numero_mesa].TMP_Etapa_Cargada.TONR(r := #cambia_registro, pt := T#10m, et => "DB920_Registro_Flujos".Mesa[#Numero_mesa].Registro["DB919_Temporizadores_Registro_flujos".Temporizadores_mesa[#Numero_mesa].NUM_REGISTRO_ACTUAL].T_Etapa_Cargada)
   END_RUNG
   // the same network as SCL:
   "DB919_Temporizadores_Registro_flujos".Temporizadores_mesa[#Numero_mesa].TMP_Etapa_Cargada.TONR(IN := NOT "DB900_Estado_Mesas".EstadoVI[#Numero_mesa].Manual AND NOT "DB900_Estado_Mesas".EstadoVI[#Numero_mesa].Paro_Blando AND NOT "DB900_Estado_Mesas".EstadoVI[#Numero_mesa].Error_Mx AND "DB900_Estado_Mesas".EstadoVI[#Numero_mesa].Etapa_Cargada,
                           R := #cambia_registro,
                           PT := T#10m,
                           ET => "DB920_Registro_Flujos".Mesa[#Numero_mesa].Registro["DB919_Temporizadores_Registro_flujos".Temporizadores_mesa[#Numero_mesa].NUM_REGISTRO_ACTUAL].T_Etapa_Cargada);
END_REGION

REGION Network 6: Temporizador Avance/Retroceso Rodillos
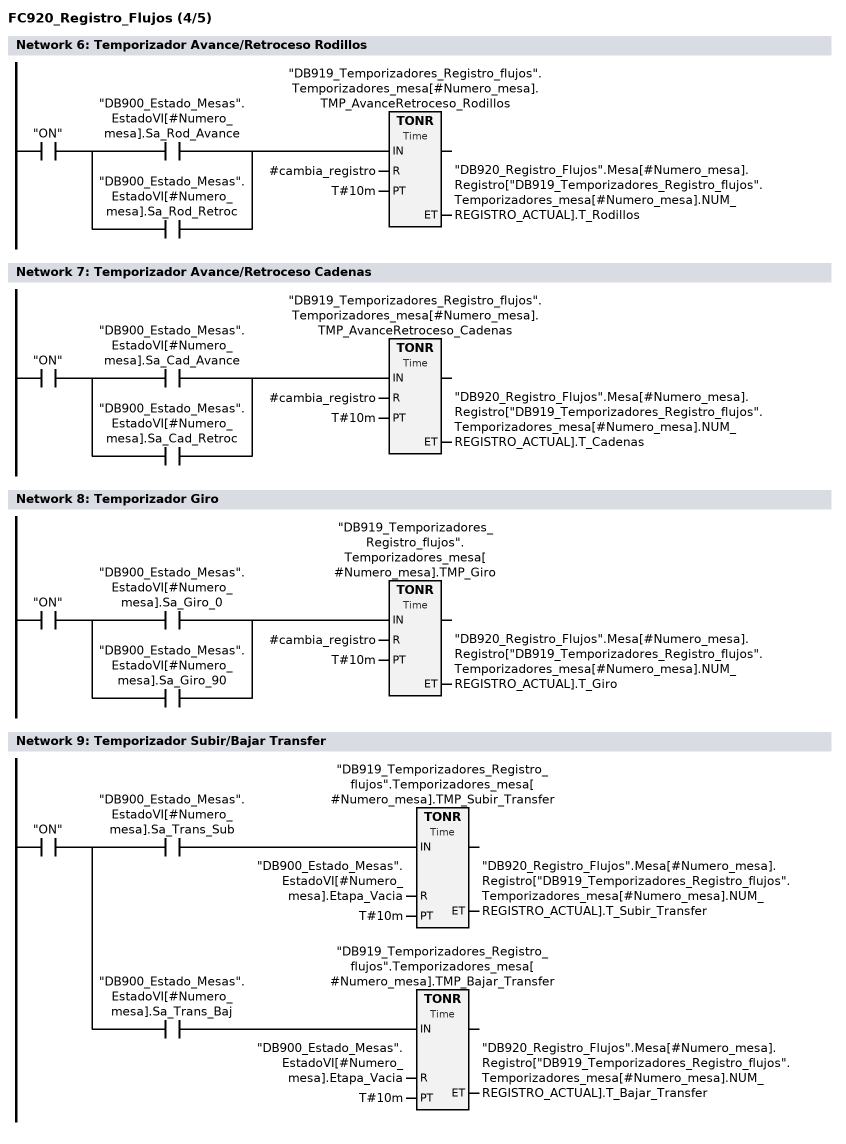
   RUNG wire#powerrail
      Contact( "ON" )
      wire#w1
      Contact( "DB900_Estado_Mesas".EstadoVI[#Numero_mesa].Sa_Rod_Avance )
      wire#w2
      { S7_Templates := "time_type := Time" } "DB919_Temporizadores_Registro_flujos".Temporizadores_mesa[#Numero_mesa].TMP_AvanceRetroceso_Rodillos.TONR(r := #cambia_registro, pt := T#10m, et => "DB920_Registro_Flujos".Mesa[#Numero_mesa].Registro["DB919_Temporizadores_Registro_flujos".Temporizadores_mesa[#Numero_mesa].NUM_REGISTRO_ACTUAL].T_Rodillos)
   END_RUNG
   RUNG wire#w1
      Contact( "DB900_Estado_Mesas".EstadoVI[#Numero_mesa].Sa_Rod_Retroc )
   END_RUNG wire#w2
   // the same network as SCL:
   "DB919_Temporizadores_Registro_flujos".Temporizadores_mesa[#Numero_mesa].TMP_AvanceRetroceso_Rodillos.TONR(IN := "ON" AND ("DB900_Estado_Mesas".EstadoVI[#Numero_mesa].Sa_Rod_Avance OR "DB900_Estado_Mesas".EstadoVI[#Numero_mesa].Sa_Rod_Retroc),
                           R := #cambia_registro,
                           PT := T#10m,
                           ET => "DB920_Registro_Flujos".Mesa[#Numero_mesa].Registro["DB919_Temporizadores_Registro_flujos".Temporizadores_mesa[#Numero_mesa].NUM_REGISTRO_ACTUAL].T_Rodillos);
END_REGION

REGION Network 7: Temporizador Avance/Retroceso Cadenas
   RUNG wire#powerrail
      Contact( "ON" )
      wire#w1
      Contact( "DB900_Estado_Mesas".EstadoVI[#Numero_mesa].Sa_Cad_Avance )
      wire#w2
      { S7_Templates := "time_type := Time" } "DB919_Temporizadores_Registro_flujos".Temporizadores_mesa[#Numero_mesa].TMP_AvanceRetroceso_Cadenas.TONR(r := #cambia_registro, pt := T#10m, et => "DB920_Registro_Flujos".Mesa[#Numero_mesa].Registro["DB919_Temporizadores_Registro_flujos".Temporizadores_mesa[#Numero_mesa].NUM_REGISTRO_ACTUAL].T_Cadenas)
   END_RUNG
   RUNG wire#w1
      Contact( "DB900_Estado_Mesas".EstadoVI[#Numero_mesa].Sa_Cad_Retroc )
   END_RUNG wire#w2
   // the same network as SCL:
   "DB919_Temporizadores_Registro_flujos".Temporizadores_mesa[#Numero_mesa].TMP_AvanceRetroceso_Cadenas.TONR(IN := "ON" AND ("DB900_Estado_Mesas".EstadoVI[#Numero_mesa].Sa_Cad_Avance OR "DB900_Estado_Mesas".EstadoVI[#Numero_mesa].Sa_Cad_Retroc),
                           R := #cambia_registro,
                           PT := T#10m,
                           ET => "DB920_Registro_Flujos".Mesa[#Numero_mesa].Registro["DB919_Temporizadores_Registro_flujos".Temporizadores_mesa[#Numero_mesa].NUM_REGISTRO_ACTUAL].T_Cadenas);
END_REGION

REGION Network 8: Temporizador Giro
   RUNG wire#powerrail
      Contact( "ON" )
      wire#w1
      Contact( "DB900_Estado_Mesas".EstadoVI[#Numero_mesa].Sa_Giro_0 )
      wire#w2
      { S7_Templates := "time_type := Time" } "DB919_Temporizadores_Registro_flujos".Temporizadores_mesa[#Numero_mesa].TMP_Giro.TONR(r := #cambia_registro, pt := T#10m, et => "DB920_Registro_Flujos".Mesa[#Numero_mesa].Registro["DB919_Temporizadores_Registro_flujos".Temporizadores_mesa[#Numero_mesa].NUM_REGISTRO_ACTUAL].T_Giro)
   END_RUNG
   RUNG wire#w1
      Contact( "DB900_Estado_Mesas".EstadoVI[#Numero_mesa].Sa_Giro_90 )
   END_RUNG wire#w2
   // the same network as SCL:
   "DB919_Temporizadores_Registro_flujos".Temporizadores_mesa[#Numero_mesa].TMP_Giro.TONR(IN := "ON" AND ("DB900_Estado_Mesas".EstadoVI[#Numero_mesa].Sa_Giro_0 OR "DB900_Estado_Mesas".EstadoVI[#Numero_mesa].Sa_Giro_90),
                           R := #cambia_registro,
                           PT := T#10m,
                           ET => "DB920_Registro_Flujos".Mesa[#Numero_mesa].Registro["DB919_Temporizadores_Registro_flujos".Temporizadores_mesa[#Numero_mesa].NUM_REGISTRO_ACTUAL].T_Giro);
END_REGION

REGION Network 9: Temporizador Subir/Bajar Transfer
   RUNG wire#powerrail
      Contact( "ON" )
      wire#w1
      Contact( "DB900_Estado_Mesas".EstadoVI[#Numero_mesa].Sa_Trans_Sub )
      { S7_Templates := "time_type := Time" } "DB919_Temporizadores_Registro_flujos".Temporizadores_mesa[#Numero_mesa].TMP_Subir_Transfer.TONR(r := "DB900_Estado_Mesas".EstadoVI[#Numero_mesa].Etapa_Vacia, pt := T#10m, et => "DB920_Registro_Flujos".Mesa[#Numero_mesa].Registro["DB919_Temporizadores_Registro_flujos".Temporizadores_mesa[#Numero_mesa].NUM_REGISTRO_ACTUAL].T_Subir_Transfer)
   END_RUNG
   RUNG wire#w1
      Contact( "DB900_Estado_Mesas".EstadoVI[#Numero_mesa].Sa_Trans_Baj )
      { S7_Templates := "time_type := Time" } "DB919_Temporizadores_Registro_flujos".Temporizadores_mesa[#Numero_mesa].TMP_Bajar_Transfer.TONR(r := "DB900_Estado_Mesas".EstadoVI[#Numero_mesa].Etapa_Vacia, pt := T#10m, et => "DB920_Registro_Flujos".Mesa[#Numero_mesa].Registro["DB919_Temporizadores_Registro_flujos".Temporizadores_mesa[#Numero_mesa].NUM_REGISTRO_ACTUAL].T_Bajar_Transfer)
   END_RUNG
   // the same network as SCL:
   "DB919_Temporizadores_Registro_flujos".Temporizadores_mesa[#Numero_mesa].TMP_Subir_Transfer.TONR(IN := "ON" AND "DB900_Estado_Mesas".EstadoVI[#Numero_mesa].Sa_Trans_Sub,
                           R := "DB900_Estado_Mesas".EstadoVI[#Numero_mesa].Etapa_Vacia,
                           PT := T#10m,
                           ET => "DB920_Registro_Flujos".Mesa[#Numero_mesa].Registro["DB919_Temporizadores_Registro_flujos".Temporizadores_mesa[#Numero_mesa].NUM_REGISTRO_ACTUAL].T_Subir_Transfer);
   "DB919_Temporizadores_Registro_flujos".Temporizadores_mesa[#Numero_mesa].TMP_Bajar_Transfer.TONR(IN := "ON" AND "DB900_Estado_Mesas".EstadoVI[#Numero_mesa].Sa_Trans_Baj,
                           R := "DB900_Estado_Mesas".EstadoVI[#Numero_mesa].Etapa_Vacia,
                           PT := T#10m,
                           ET => "DB920_Registro_Flujos".Mesa[#Numero_mesa].Registro["DB919_Temporizadores_Registro_flujos".Temporizadores_mesa[#Numero_mesa].NUM_REGISTRO_ACTUAL].T_Bajar_Transfer);
END_REGION

REGION Network 10: Temporizador TOTAL
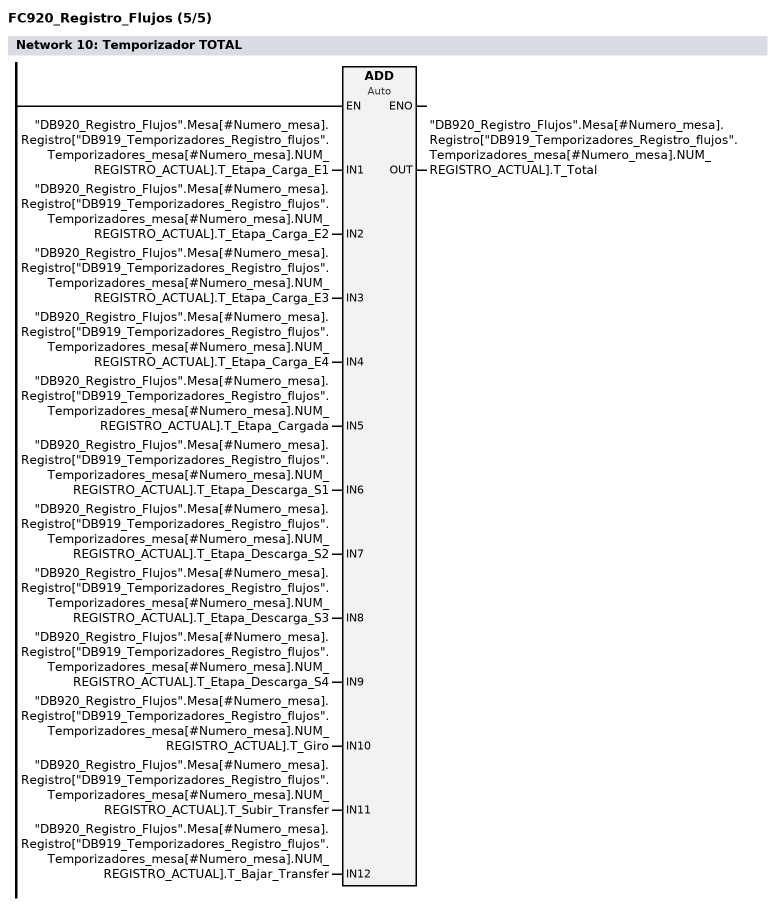
   RUNG wire#powerrail
      Add(in1 := "DB920_Registro_Flujos".Mesa[#Numero_mesa].Registro["DB919_Temporizadores_Registro_flujos".Temporizadores_mesa[#Numero_mesa].NUM_REGISTRO_ACTUAL].T_Etapa_Carga_E1, in2 := "DB920_Registro_Flujos".Mesa[#Numero_mesa].Registro["DB919_Temporizadores_Registro_flujos".Temporizadores_mesa[#Numero_mesa].NUM_REGISTRO_ACTUAL].T_Etapa_Carga_E2, in3 := "DB920_Registro_Flujos".Mesa[#Numero_mesa].Registro["DB919_Temporizadores_Registro_flujos".Temporizadores_mesa[#Numero_mesa].NUM_REGISTRO_ACTUAL].T_Etapa_Carga_E3, in4 := "DB920_Registro_Flujos".Mesa[#Numero_mesa].Registro["DB919_Temporizadores_Registro_flujos".Temporizadores_mesa[#Numero_mesa].NUM_REGISTRO_ACTUAL].T_Etapa_Carga_E4, in5 := "DB920_Registro_Flujos".Mesa[#Numero_mesa].Registro["DB919_Temporizadores_Registro_flujos".Temporizadores_mesa[#Numero_mesa].NUM_REGISTRO_ACTUAL].T_Etapa_Cargada, in6 := "DB920_Registro_Flujos".Mesa[#Numero_mesa].Registro["DB919_Temporizadores_Registro_flujos".Temporizadores_mesa[#Numero_mesa].NUM_REGISTRO_ACTUAL].T_Etapa_Descarga_S1, in7 := "DB920_Registro_Flujos".Mesa[#Numero_mesa].Registro["DB919_Temporizadores_Registro_flujos".Temporizadores_mesa[#Numero_mesa].NUM_REGISTRO_ACTUAL].T_Etapa_Descarga_S2, in8 := "DB920_Registro_Flujos".Mesa[#Numero_mesa].Registro["DB919_Temporizadores_Registro_flujos".Temporizadores_mesa[#Numero_mesa].NUM_REGISTRO_ACTUAL].T_Etapa_Descarga_S3, in9 := "DB920_Registro_Flujos".Mesa[#Numero_mesa].Registro["DB919_Temporizadores_Registro_flujos".Temporizadores_mesa[#Numero_mesa].NUM_REGISTRO_ACTUAL].T_Etapa_Descarga_S4, in10 := "DB920_Registro_Flujos".Mesa[#Numero_mesa].Registro["DB919_Temporizadores_Registro_flujos".Temporizadores_mesa[#Numero_mesa].NUM_REGISTRO_ACTUAL].T_Giro, in11 := "DB920_Registro_Flujos".Mesa[#Numero_mesa].Registro["DB919_Temporizadores_Registro_flujos".Temporizadores_mesa[#Numero_mesa].NUM_REGISTRO_ACTUAL].T_Subir_Transfer, in12 := "DB920_Registro_Flujos".Mesa[#Numero_mesa].Registro["DB919_Temporizadores_Registro_flujos".Temporizadores_mesa[#Numero_mesa].NUM_REGISTRO_ACTUAL].T_Bajar_Transfer, out => "DB920_Registro_Flujos".Mesa[#Numero_mesa].Registro["DB919_Temporizadores_Registro_flujos".Temporizadores_mesa[#Numero_mesa].NUM_REGISTRO_ACTUAL].T_Total)
   END_RUNG
   // the same network as SCL:
   "DB920_Registro_Flujos".Mesa[#Numero_mesa].Registro["DB919_Temporizadores_Registro_flujos".Temporizadores_mesa[#Numero_mesa].NUM_REGISTRO_ACTUAL].T_Total := "DB920_Registro_Flujos".Mesa[#Numero_mesa].Registro["DB919_Temporizadores_Registro_flujos".Temporizadores_mesa[#Numero_mesa].NUM_REGISTRO_ACTUAL].T_Etapa_Carga_E1 + "DB920_Registro_Flujos".Mesa[#Numero_mesa].Registro["DB919_Temporizadores_Registro_flujos".Temporizadores_mesa[#Numero_mesa].NUM_REGISTRO_ACTUAL].T_Etapa_Carga_E2 + "DB920_Registro_Flujos".Mesa[#Numero_mesa].Registro["DB919_Temporizadores_Registro_flujos".Temporizadores_mesa[#Numero_mesa].NUM_REGISTRO_ACTUAL].T_Etapa_Carga_E3 + "DB920_Registro_Flujos".Mesa[#Numero_mesa].Registro["DB919_Temporizadores_Registro_flujos".Temporizadores_mesa[#Numero_mesa].NUM_REGISTRO_ACTUAL].T_Etapa_Carga_E4 + "DB920_Registro_Flujos".Mesa[#Numero_mesa].Registro["DB919_Temporizadores_Registro_flujos".Temporizadores_mesa[#Numero_mesa].NUM_REGISTRO_ACTUAL].T_Etapa_Cargada + "DB920_Registro_Flujos".Mesa[#Numero_mesa].Registro["DB919_Temporizadores_Registro_flujos".Temporizadores_mesa[#Numero_mesa].NUM_REGISTRO_ACTUAL].T_Etapa_Descarga_S1 + "DB920_Registro_Flujos".Mesa[#Numero_mesa].Registro["DB919_Temporizadores_Registro_flujos".Temporizadores_mesa[#Numero_mesa].NUM_REGISTRO_ACTUAL].T_Etapa_Descarga_S2 + "DB920_Registro_Flujos".Mesa[#Numero_mesa].Registro["DB919_Temporizadores_Registro_flujos".Temporizadores_mesa[#Numero_mesa].NUM_REGISTRO_ACTUAL].T_Etapa_Descarga_S3 + "DB920_Registro_Flujos".Mesa[#Numero_mesa].Registro["DB919_Temporizadores_Registro_flujos".Temporizadores_mesa[#Numero_mesa].NUM_REGISTRO_ACTUAL].T_Etapa_Descarga_S4 + "DB920_Registro_Flujos".Mesa[#Numero_mesa].Registro["DB919_Temporizadores_Registro_flujos".Temporizadores_mesa[#Numero_mesa].NUM_REGISTRO_ACTUAL].T_Giro + "DB920_Registro_Flujos".Mesa[#Numero_mesa].Registro["DB919_Temporizadores_Registro_flujos".Temporizadores_mesa[#Numero_mesa].NUM_REGISTRO_ACTUAL].T_Subir_Transfer + "DB920_Registro_Flujos".Mesa[#Numero_mesa].Registro["DB919_Temporizadores_Registro_flujos".Temporizadores_mesa[#Numero_mesa].NUM_REGISTRO_ACTUAL].T_Bajar_Transfer;
END_REGION
END_FUNCTION

FUNCTION "FC983_CTRL_SmartMotor_3AD_1AT" : Void   // FC983, LAD
{ S7_Optimized_Access := 'TRUE' }
// stored: AutoNumber false, SetENOAutomatically false
   VAR_INPUT
      Avance : Bool;
      Retroceso_Manual : Bool;
      Vel_Rapida : Bool;
      Vel_Manual : Bool;
      T_Decel : UDInt;   // base tiempo ms
   END_VAR
   VAR_OUTPUT
      Av_Ret_Tx : Bool;
      DO1 : Bool;
      DO2 : Bool;
      DO3 : Bool;
   END_VAR
   VAR_IN_OUT
      TMP_Deceleracion : UDInt;
   END_VAR
   VAR_TEMP
      Parado_del_todo : Bool;
   END_VAR
BEGIN

REGION Network 1: Activación DI1 del Smart Motor
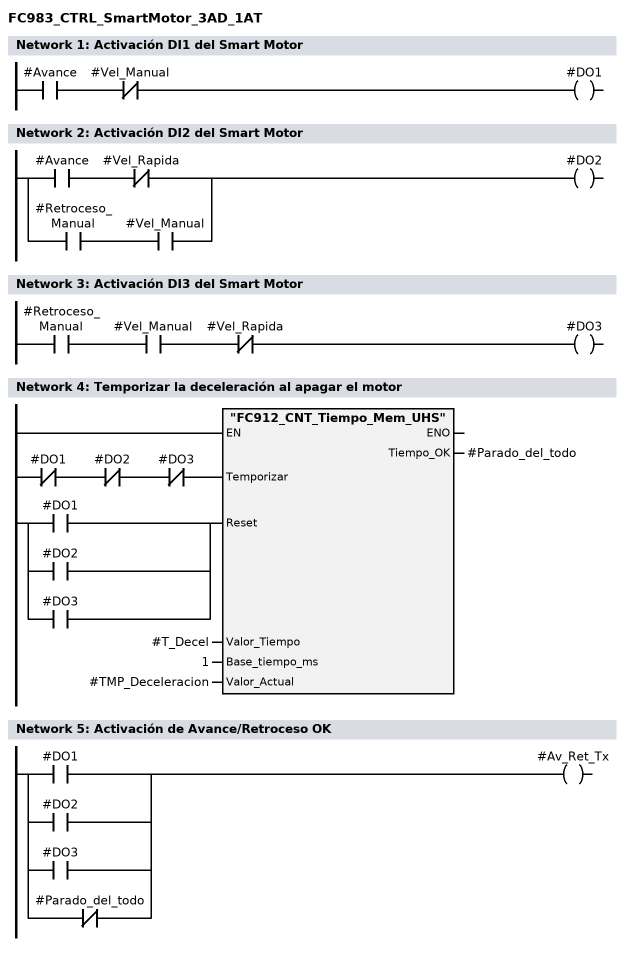
   RUNG wire#powerrail
      Contact( #Avance )
      I_Contact( #Vel_Manual )
      Coil( #DO1 )
   END_RUNG
   // the same network as SCL:
   #DO1 := #Avance AND NOT #Vel_Manual;
END_REGION

REGION Network 2: Activación DI2 del Smart Motor
   RUNG wire#powerrail
      Contact( #Avance )
      I_Contact( #Vel_Rapida )
      wire#w1
      Coil( #DO2 )
   END_RUNG
   RUNG wire#powerrail
      Contact( #Retroceso_Manual )
      Contact( #Vel_Manual )
   END_RUNG wire#w1
   // the same network as SCL:
   #DO2 := (#Avance AND NOT #Vel_Rapida) OR (#Retroceso_Manual AND #Vel_Manual);
END_REGION

REGION Network 3: Activación DI3 del Smart Motor
   RUNG wire#powerrail
      Contact( #Retroceso_Manual )
      Contact( #Vel_Manual )
      I_Contact( #Vel_Rapida )
      Coil( #DO3 )
   END_RUNG
   // the same network as SCL:
   #DO3 := #Retroceso_Manual AND #Vel_Manual AND NOT #Vel_Rapida;
END_REGION

REGION Network 4: Temporizar la deceleración al apagar el motor
   RUNG wire#powerrail
      "FC912_CNT_Tiempo_Mem_UHS"(Temporizar := wire#w1, Reset := wire#w2, Valor_Tiempo := #T_Decel, Base_tiempo_ms := 1, Valor_Actual := #TMP_Deceleracion, Tiempo_OK => #Parado_del_todo)
   END_RUNG
   RUNG wire#powerrail
      I_Contact( #DO1 )
      I_Contact( #DO2 )
      I_Contact( #DO3 )
   END_RUNG wire#w1
   RUNG wire#powerrail
      Contact( #DO1 )
   END_RUNG wire#w2
   RUNG wire#powerrail
      Contact( #DO2 )
   END_RUNG wire#w2
   RUNG wire#powerrail
      Contact( #DO3 )
   END_RUNG wire#w2
   // the same network as SCL:
   "FC912_CNT_Tiempo_Mem_UHS"(Temporizar := NOT #DO1 AND NOT #DO2 AND NOT #DO3,
                           Reset := #DO1 OR #DO2 OR #DO3,
                           Valor_Tiempo := #T_Decel,
                           Base_tiempo_ms := 1,
                           Valor_Actual := #TMP_Deceleracion,
                           Tiempo_OK => #Parado_del_todo);
END_REGION

REGION Network 5: Activación de Avance/Retroceso OK
   RUNG wire#powerrail
      Contact( #DO1 )
      wire#w1
      Coil( #Av_Ret_Tx )
   END_RUNG
   RUNG wire#powerrail
      Contact( #DO2 )
   END_RUNG wire#w1
   RUNG wire#powerrail
      Contact( #DO3 )
   END_RUNG wire#w1
   RUNG wire#powerrail
      I_Contact( #Parado_del_todo )
   END_RUNG wire#w1
   // the same network as SCL:
   #Av_Ret_Tx := #DO1 OR #DO2 OR #DO3 OR NOT #Parado_del_todo;
END_REGION
END_FUNCTION

FUNCTION "FC9_JDT_Adaptacion" : Void   // FC9, LAD
{ S7_Optimized_Access := 'TRUE' }
// stored: AutoNumber false, SetENOAutomatically false
   VAR_INPUT
      Zona : UInt;   // Numero de Zona
      INP_Pul_TLuces : Bool;
      Jdt_Marcha : Bool;
      JdT_Paro : Bool;
      JdT_Reset : Bool;
      JdT_EmiOK : Bool;
   END_VAR
   VAR_OUTPUT
      L_Verde : Bool;
      L_Naranja : Bool;
      L_Rojo : Bool;
      PLC_Automatico : Bool;
      PLC_Manual : Bool;
      PLC_Marcha : Bool;
      PLC_Paro : Bool;
      PLC_Error : Bool;
      PLC_Reset_OK : Bool;
      PLC_Reset_NOK : Bool;
      PLC_RecepOK : Bool;
   END_VAR
   VAR_IN_OUT
      CodigoError : Word;
   END_VAR
   VAR_TEMP
      MesaEnError : UInt;
   END_VAR
BEGIN

NETWORK
TITLE = INICIALIZAR

NETWORK
TITLE = CODIGO DE ERROR - DE ZONA
/////////////////////////////////////////////////////////////////////////////////////
////////////////////////////////////////////////////////////////////////////////////
////////////////////////////////////////////////////////////////////////////////////
/// --- Codigo de Error De Zona Dos Digitos -- 9x EE
      L     0;  // Inicializa el Codigo de Error
      T     #CodigoError;

      SET;  // Existe Error de Zona ?
      AN    "DB840_Emision".DispoArmario[#Zona].Protocolo.Error;
      JC    Final_ErrorDeZona;

/// --- Primer Digito - Error
      L     "DB840_Emision".DispoArmario[#Zona].Error;
      L     10;
      MOD;
      T     #CodigoError;

/// --- Segundo Digito - Error
      L     "DB840_Emision".DispoArmario[#Zona].Error;
      L     10;
      /D;
      L     10;
      MOD;
      SLD   4;
      L     #CodigoError;
      OW;
      T     #CodigoError;

/// --- Tercer Digito - Numero de Zona
      L     #Zona;
      SLD   8;
      L     #CodigoError;
      OW;
      T     #CodigoError;

/// --- Cuarto Digito - Indicacion De Zona
      L     w#16#9000;
      L     #CodigoError;
      OW;
      T     #CodigoError;

/// --- Final de Codificacion del Error de Zona
Final_ErrorDeZona:NOP   0;



NETWORK
TITLE = CODIGO DE ERROR - DE MESA
/////////////////////////////////////////////////////////////////////////////////////
////////////////////////////////////////////////////////////////////////////////////
////////////////////////////////////////////////////////////////////////////////////
/// --- Codigo de Error De Mesa -- 6 MMMM
      SET;  // Existe Error de Zona ?
      A     "DB840_Emision".DispoArmario[#Zona].Protocolo.Error;
      JC    Final_ErrorDeMesa;

      SET;  // Existe Error de Mesa ?
      AN    "DB901_Estado_Zonas".EstadoZona[#Zona].VariablesInternas.MesasError;
      JC    Final_ErrorDeMesa;

/// --- Numero de Mesa en Error
      L     0;
      T     #MesaEnError;
InicioBucle_BusquedaDeMesaEnError:NOP   0;
      L     "CTE_MaxMesas";  // - Final del Numero de Mesas ?
      L     #MesaEnError;
      <=I;
      JC    FinalBucle_BusquedaDeMesaEnError;

      L     #MesaEnError;
      L     1;
      +I;
      T     #MesaEnError;

      SET;  /// Mesa de la Zona (0)
      L     #Zona;
      L     "DB914_Conf_Mesas_DeZona".MesasDeZona[#MesaEnError, 0].ZonaPerteneceMesa;
      ==I;
      JC    MesaEncontrada_BusquedaDeMEsaEnError;

      SET;  /// Mesa de la Zona (1)
      L     #Zona;
      L     "DB914_Conf_Mesas_DeZona".MesasDeZona[#MesaEnError, 1].ZonaPerteneceMesa;
      ==I;
      JC    MesaEncontrada_BusquedaDeMEsaEnError;

      SET;  /// Mesa de la Zona (2)
      L     #Zona;
      L     "DB914_Conf_Mesas_DeZona".MesasDeZona[#MesaEnError, 2].ZonaPerteneceMesa;
      ==I;
      JC    MesaEncontrada_BusquedaDeMEsaEnError;

      SET;  /// Mesa de la Zona (3)
      L     #Zona;
      L     "DB914_Conf_Mesas_DeZona".MesasDeZona[#MesaEnError, 3].ZonaPerteneceMesa;
      ==I;
      JC    MesaEncontrada_BusquedaDeMEsaEnError;

      SET;  /// Mesa de la Zona (4)
      L     #Zona;
      L     "DB914_Conf_Mesas_DeZona".MesasDeZona[#MesaEnError, 4].ZonaPerteneceMesa;
      ==I;
      JC    MesaEncontrada_BusquedaDeMEsaEnError;

      JU    InicioBucle_BusquedaDeMesaEnError;

MesaEncontrada_BusquedaDeMEsaEnError:NOP   0;
      SET;  // - Mesa o Maquina en Error
      A     "DB902_Estado_ZonaMesa".EstadoMesas[#MesaEnError].Error_CBx;
      O     "DB903_Estado_ZonaMaquina".EstadoMaquina[#MesaEnError].Error_CBx;
      JC    FinalBucle_BusquedaDeMesaEnError;

      JU    InicioBucle_BusquedaDeMesaEnError;

////////////////////////////////////////////////////////////////////////////////////
FinalBucle_BusquedaDeMesaEnError:NOP   0;

/// --- Primer Digito - Mesa
      L     #MesaEnError;
      L     10;
      MOD;
      T     #CodigoError;

/// --- Segundo Digito - Mesa
      L     #MesaEnError;
      L     10;
      /D;
      L     10;
      MOD;
      SLD   4;
      L     #CodigoError;
      OW;
      T     #CodigoError;

/// --- Tercer Digito - Mesa
      L     #MesaEnError;
      L     100;
      /D;
      L     10;
      MOD;
      SLD   8;
      L     #CodigoError;
      OW;
      T     #CodigoError;

/// --- Cuarto Digito - Indicacion De Mesa
      L     w#16#6000;
      L     #CodigoError;
      OW;
      T     #CodigoError;

/// --- Final de Codificacion del Error de Zona
Final_ErrorDeMesa:NOP   0;



NETWORK
TITLE = EMISION DE LA ZONA
/////////////////////////////////////////////////////////////////////////////////////
////////////////////////////////////////////////////////////////////////////////////
////////////////////////////////////////////////////////////////////////////////////
/// --- COMPROBAR si esta con el JdT Antiguo
      SET;
      AN    "Activar_JdTAntiguo";
      JC    Final_EmisionZona;


/////////////////////////////////////////////////////////////////////////////////////
////////////////////////////////////////////////////////////////////////////////////
////////////////////////////////////////////////////////////////////////////////////
/// --- Automatico / Manual
      SET;
      A     "DB840_Emision".DispoArmario[#Zona].Protocolo.Automatico;
      =     #PLC_Automatico;
      SET;
      A     "DB840_Emision".DispoArmario[#Zona].Protocolo.Manual;
      =     #PLC_Manual;


/////////////////////////////////////////////////////////////////////////////////////
////////////////////////////////////////////////////////////////////////////////////
////////////////////////////////////////////////////////////////////////////////////
/// --- Marcha / Paro / ErrorPLC
      SET;
      A     "DB840_Emision".DispoArmario[#Zona].Protocolo.Marcha;
      =     #PLC_Marcha;
      SET;
      A     "DB840_Emision".DispoArmario[#Zona].Protocolo.Paro;
      =     #PLC_Paro;
      SET;
      A     "DB840_Emision".DispoArmario[#Zona].Protocolo.Error;
      O     "DB901_Estado_Zonas".EstadoZona[#Zona].VariablesInternas.MesasError;
      =     #PLC_Error;

/////////////////////////////////////////////////////////////////////////////////////
////////////////////////////////////////////////////////////////////////////////////
////////////////////////////////////////////////////////////////////////////////////
/// --- Reset
      SET;
      A     "DB840_Emision".DispoArmario[#Zona].Protocolo.ResetOK;
      =     #PLC_Reset_OK;
      SET;
      A     "DB840_Emision".DispoArmario[#Zona].Protocolo.ResetNOK;
      =     #PLC_Reset_NOK;

/////////////////////////////////////////////////////////////////////////////////////
////////////////////////////////////////////////////////////////////////////////////
////////////////////////////////////////////////////////////////////////////////////
/// --- Comunicacion
      SET;
      A     "DB840_Emision".DispoArmario[#Zona].Protocolo.RecepOK;
      =     #PLC_RecepOK;


/////////////////////////////////////////////////////////////////////////////////////
////////////////////////////////////////////////////////////////////////////////////
////////////////////////////////////////////////////////////////////////////////////
/// --- FINAL de la EMISION DE LA ZONA
Final_EmisionZona:NOP   0;



NETWORK
TITLE = RECEPCION DE LA ZONA
/////////////////////////////////////////////////////////////////////////////////////
////////////////////////////////////////////////////////////////////////////////////
////////////////////////////////////////////////////////////////////////////////////
/// --- COMPROBAR si esta con el JdT Antiguo
      SET;
      AN    "Activar_JdTAntiguo";
      JC    Final_RecepcionZona;


/////////////////////////////////////////////////////////////////////////////////////
/////////////////////////////////////////////////////////////////////////////////////
/////////////////////////////////////////////////////////////////////////////////////
/// --- Ordenes
      SET;
      A     #Jdt_Marcha;
      =     "DB841_Recepcion".DispoArmario[#Zona].Protocolo.Marcha;
      SET;
      A     #JdT_Paro;
      =     "DB841_Recepcion".DispoArmario[#Zona].Protocolo.Paro;
      SET;
      A     #JdT_Reset;
      =     "DB841_Recepcion".DispoArmario[#Zona].Protocolo.Reset;

/////////////////////////////////////////////////////////////////////////////////////
////////////////////////////////////////////////////////////////////////////////////
////////////////////////////////////////////////////////////////////////////////////
/// --- Comunicacion
      SET;
      A     #JdT_EmiOK;
      =     "DB841_Recepcion".DispoArmario[#Zona].Protocolo.EmiOK;


/////////////////////////////////////////////////////////////////////////////////////
////////////////////////////////////////////////////////////////////////////////////
////////////////////////////////////////////////////////////////////////////////////
/// --- FINAL de la RECEPCION DE LA ZONA
Final_RecepcionZona:NOP   0;



REGION Network 6: SALIDAS - Baliza VERDE
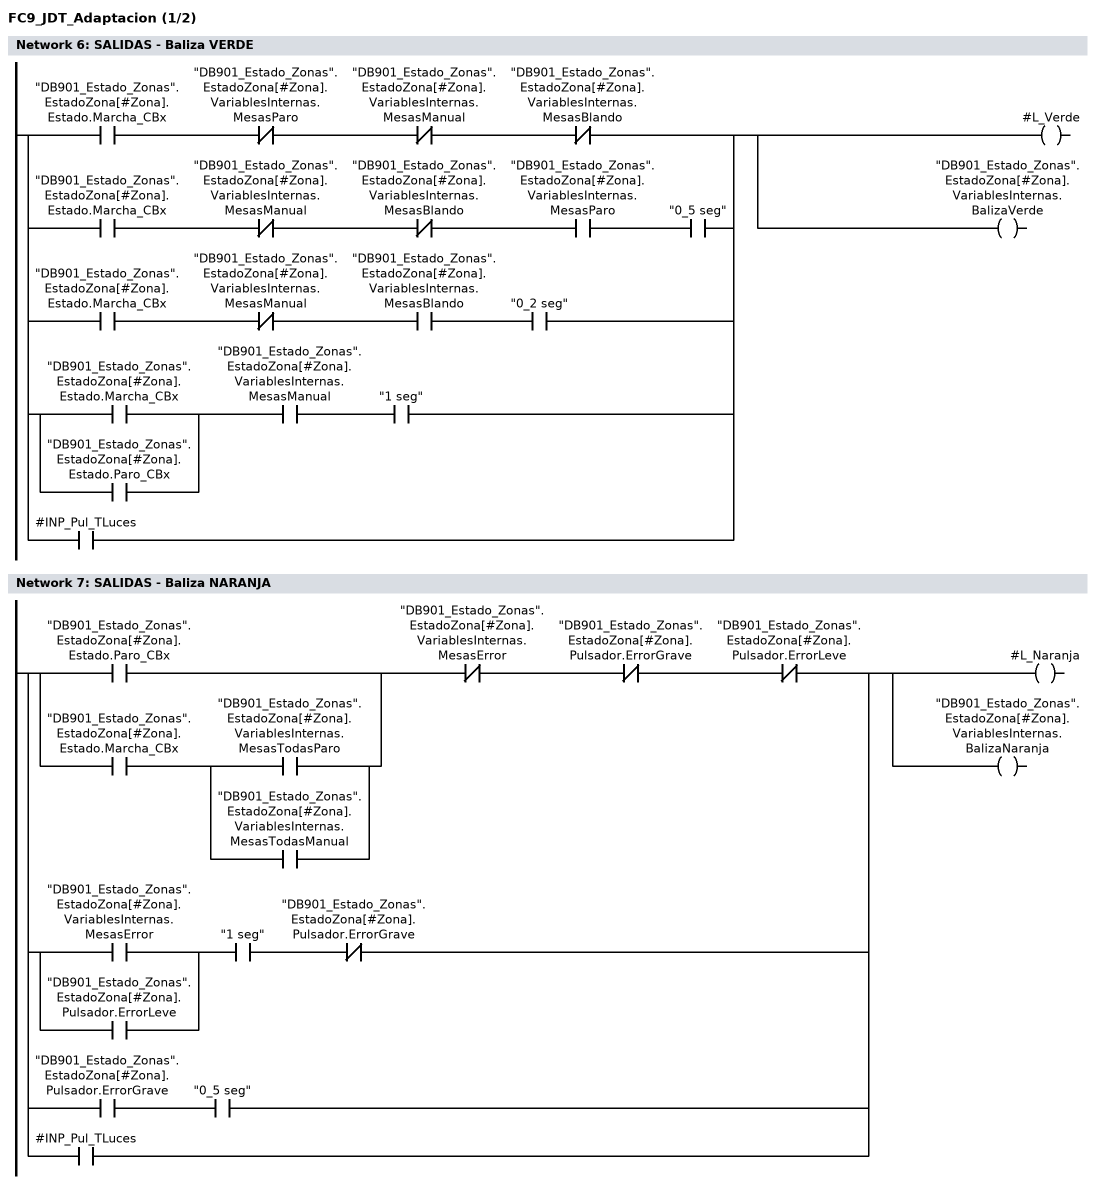
   RUNG wire#powerrail
      Contact( "DB901_Estado_Zonas".EstadoZona[#Zona].Estado.Marcha_CBx )
      I_Contact( "DB901_Estado_Zonas".EstadoZona[#Zona].VariablesInternas.MesasParo )
      I_Contact( "DB901_Estado_Zonas".EstadoZona[#Zona].VariablesInternas.MesasManual )
      I_Contact( "DB901_Estado_Zonas".EstadoZona[#Zona].VariablesInternas.MesasBlando )
      wire#w1
      Coil( #L_Verde )
   END_RUNG
   RUNG wire#powerrail
      Contact( "DB901_Estado_Zonas".EstadoZona[#Zona].Estado.Marcha_CBx )
      I_Contact( "DB901_Estado_Zonas".EstadoZona[#Zona].VariablesInternas.MesasManual )
      I_Contact( "DB901_Estado_Zonas".EstadoZona[#Zona].VariablesInternas.MesasBlando )
      Contact( "DB901_Estado_Zonas".EstadoZona[#Zona].VariablesInternas.MesasParo )
      Contact( "0_5 seg" )
   END_RUNG wire#w1
   RUNG wire#powerrail
      Contact( "DB901_Estado_Zonas".EstadoZona[#Zona].Estado.Marcha_CBx )
      I_Contact( "DB901_Estado_Zonas".EstadoZona[#Zona].VariablesInternas.MesasManual )
      Contact( "DB901_Estado_Zonas".EstadoZona[#Zona].VariablesInternas.MesasBlando )
      Contact( "0_2 seg" )
   END_RUNG wire#w1
   RUNG wire#powerrail
      Contact( "DB901_Estado_Zonas".EstadoZona[#Zona].Estado.Marcha_CBx )
      wire#w2
      Contact( "DB901_Estado_Zonas".EstadoZona[#Zona].VariablesInternas.MesasManual )
      Contact( "1 seg" )
   END_RUNG wire#w1
   RUNG wire#powerrail
      Contact( "DB901_Estado_Zonas".EstadoZona[#Zona].Estado.Paro_CBx )
   END_RUNG wire#w2
   RUNG wire#powerrail
      Contact( #INP_Pul_TLuces )
   END_RUNG wire#w1
   RUNG wire#w1
      Coil( "DB901_Estado_Zonas".EstadoZona[#Zona].VariablesInternas.BalizaVerde )
   END_RUNG
   // the same network as SCL:
   #L_Verde := ("DB901_Estado_Zonas".EstadoZona[#Zona].Estado.Marcha_CBx AND NOT "DB901_Estado_Zonas".EstadoZona[#Zona].VariablesInternas.MesasParo AND NOT "DB901_Estado_Zonas".EstadoZona[#Zona].VariablesInternas.MesasManual AND NOT "DB901_Estado_Zonas".EstadoZona[#Zona].VariablesInternas.MesasBlando) OR ("DB901_Estado_Zonas".EstadoZona[#Zona].Estado.Marcha_CBx AND NOT "DB901_Estado_Zonas".EstadoZona[#Zona].VariablesInternas.MesasManual AND NOT "DB901_Estado_Zonas".EstadoZona[#Zona].VariablesInternas.MesasBlando AND "DB901_Estado_Zonas".EstadoZona[#Zona].VariablesInternas.MesasParo AND "0_5 seg") OR ("DB901_Estado_Zonas".EstadoZona[#Zona].Estado.Marcha_CBx AND NOT "DB901_Estado_Zonas".EstadoZona[#Zona].VariablesInternas.MesasManual AND "DB901_Estado_Zonas".EstadoZona[#Zona].VariablesInternas.MesasBlando AND "0_2 seg") OR (("DB901_Estado_Zonas".EstadoZona[#Zona].Estado.Marcha_CBx OR "DB901_Estado_Zonas".EstadoZona[#Zona].Estado.Paro_CBx) AND "DB901_Estado_Zonas".EstadoZona[#Zona].VariablesInternas.MesasManual AND "1 seg") OR #INP_Pul_TLuces;
   "DB901_Estado_Zonas".EstadoZona[#Zona].VariablesInternas.BalizaVerde := #L_Verde;
END_REGION

REGION Network 7: SALIDAS - Baliza NARANJA
   RUNG wire#powerrail
      Contact( "DB901_Estado_Zonas".EstadoZona[#Zona].Estado.Paro_CBx )
      wire#w1
      I_Contact( "DB901_Estado_Zonas".EstadoZona[#Zona].VariablesInternas.MesasError )
      I_Contact( "DB901_Estado_Zonas".EstadoZona[#Zona].Pulsador.ErrorGrave )
      I_Contact( "DB901_Estado_Zonas".EstadoZona[#Zona].Pulsador.ErrorLeve )
      wire#w3
      Coil( #L_Naranja )
   END_RUNG
   RUNG wire#powerrail
      Contact( "DB901_Estado_Zonas".EstadoZona[#Zona].Estado.Marcha_CBx )
      wire#w2
      Contact( "DB901_Estado_Zonas".EstadoZona[#Zona].VariablesInternas.MesasTodasParo )
   END_RUNG wire#w1
   RUNG wire#w2
      Contact( "DB901_Estado_Zonas".EstadoZona[#Zona].VariablesInternas.MesasTodasManual )
   END_RUNG wire#w1
   RUNG wire#powerrail
      Contact( "DB901_Estado_Zonas".EstadoZona[#Zona].VariablesInternas.MesasError )
      wire#w4
      Contact( "1 seg" )
      I_Contact( "DB901_Estado_Zonas".EstadoZona[#Zona].Pulsador.ErrorGrave )
   END_RUNG wire#w3
   RUNG wire#powerrail
      Contact( "DB901_Estado_Zonas".EstadoZona[#Zona].Pulsador.ErrorLeve )
   END_RUNG wire#w4
   RUNG wire#powerrail
      Contact( "DB901_Estado_Zonas".EstadoZona[#Zona].Pulsador.ErrorGrave )
      Contact( "0_5 seg" )
   END_RUNG wire#w3
   RUNG wire#powerrail
      Contact( #INP_Pul_TLuces )
   END_RUNG wire#w3
   RUNG wire#w3
      Coil( "DB901_Estado_Zonas".EstadoZona[#Zona].VariablesInternas.BalizaNaranja )
   END_RUNG
   // the same network as SCL:
   #L_Naranja := (("DB901_Estado_Zonas".EstadoZona[#Zona].Estado.Paro_CBx OR ("DB901_Estado_Zonas".EstadoZona[#Zona].Estado.Marcha_CBx AND ("DB901_Estado_Zonas".EstadoZona[#Zona].VariablesInternas.MesasTodasParo OR "DB901_Estado_Zonas".EstadoZona[#Zona].VariablesInternas.MesasTodasManual))) AND NOT "DB901_Estado_Zonas".EstadoZona[#Zona].VariablesInternas.MesasError AND NOT "DB901_Estado_Zonas".EstadoZona[#Zona].Pulsador.ErrorGrave AND NOT "DB901_Estado_Zonas".EstadoZona[#Zona].Pulsador.ErrorLeve) OR (("DB901_Estado_Zonas".EstadoZona[#Zona].VariablesInternas.MesasError OR "DB901_Estado_Zonas".EstadoZona[#Zona].Pulsador.ErrorLeve) AND "1 seg" AND NOT "DB901_Estado_Zonas".EstadoZona[#Zona].Pulsador.ErrorGrave) OR ("DB901_Estado_Zonas".EstadoZona[#Zona].Pulsador.ErrorGrave AND "0_5 seg") OR #INP_Pul_TLuces;
   "DB901_Estado_Zonas".EstadoZona[#Zona].VariablesInternas.BalizaNaranja := #L_Naranja;
END_REGION

